DATA_BLOCK "DB_M256A_Scada"
{ DB_Accessible_From_OPC_UA := 'FALSE' ;
 DB_Accessible_From_Webserver := 'FALSE' ;
 S7_Optimized_Access := 'FALSE' }
VERSION : 0.1
NON_RETAIN
   STRUCT
      tAlm : Struct   // HMI Alarms
         tE { ExternalWritable := 'False'} : Struct
            x0 { ExternalWritable := 'False'} : Bool;
            x1 { ExternalWritable := 'False'} : Bool;
            x2 { ExternalWritable := 'False'} : Bool;
            x3 { ExternalWritable := 'False'} : Bool;
            x4 { ExternalWritable := 'False'} : Bool;
            x5 { ExternalWritable := 'False'} : Bool;
            x6 { ExternalWritable := 'False'} : Bool;
            x7 { ExternalWritable := 'False'} : Bool;
            x8 { ExternalWritable := 'False'} : Bool;
            x9 { ExternalWritable := 'False'} : Bool;
            x10 { ExternalWritable := 'False'} : Bool;
            x11 { ExternalWritable := 'False'} : Bool;
            x12 { ExternalWritable := 'False'} : Bool;
            x13 { ExternalWritable := 'False'} : Bool;
            x14 { ExternalWritable := 'False'} : Bool;
            x15 { ExternalWritable := 'False'} : Bool;
            x16 { ExternalWritable := 'False'} : Bool;
            x17 { ExternalWritable := 'False'} : Bool;
            x18 { ExternalWritable := 'False'} : Bool;
            x19 { ExternalWritable := 'False'} : Bool;
            x20 { ExternalWritable := 'False'} : Bool;
            x21 { ExternalWritable := 'False'} : Bool;
            x22 { ExternalWritable := 'False'} : Bool;
            x23 { ExternalWritable := 'False'} : Bool;
            x24 { ExternalWritable := 'False'} : Bool;
            x25 { ExternalWritable := 'False'} : Bool;
            x26 { ExternalWritable := 'False'} : Bool;
            x27 { ExternalWritable := 'False'} : Bool;
            x28 { ExternalWritable := 'False'} : Bool;
            x29 { ExternalWritable := 'False'} : Bool;
            x30 { ExternalWritable := 'False'} : Bool;
            x31 { ExternalWritable := 'False'} : Bool;
         END_STRUCT;
         tS { ExternalWritable := 'False'} : Struct
            tS0 { ExternalWritable := 'False'} : Struct
               x0 { ExternalWritable := 'False'} : Bool;   // Head#1 carriage not in working position
               x1 { ExternalWritable := 'False'} : Bool;   //
               x2 { ExternalWritable := 'False'} : Bool;
               x3 { ExternalWritable := 'False'} : Bool;
               x4 { ExternalWritable := 'False'} : Bool;
               x5 { ExternalWritable := 'False'} : Bool;
               x6 { ExternalWritable := 'False'} : Bool;
               x7 { ExternalWritable := 'False'} : Bool;
               x8 { ExternalWritable := 'False'} : Bool;
               x9 { ExternalWritable := 'False'} : Bool;   // Head#2carriage not in working position
               x10 { ExternalWritable := 'False'} : Bool;
               x11 { ExternalWritable := 'False'} : Bool;
               x12 { ExternalWritable := 'False'} : Bool;
               x13 { ExternalWritable := 'False'} : Bool;
               x14 { ExternalWritable := 'False'} : Bool;
               x15 { ExternalWritable := 'False'} : Bool;
               x16 { ExternalWritable := 'False'} : Bool;
               x17 { ExternalWritable := 'False'} : Bool;
               x18 { ExternalWritable := 'False'} : Bool;   // Head#3carriage not in working position
               x19 { ExternalWritable := 'False'} : Bool;
               x20 { ExternalWritable := 'False'} : Bool;
               x21 { ExternalWritable := 'False'} : Bool;
               x22 { ExternalWritable := 'False'} : Bool;
               x23 { ExternalWritable := 'False'} : Bool;
               x24 { ExternalWritable := 'False'} : Bool;
               x25 { ExternalWritable := 'False'} : Bool;
               x26 { ExternalWritable := 'False'} : Bool;
               x27 { ExternalWritable := 'False'} : Bool;
               x28 { ExternalWritable := 'False'} : Bool;
               x29 { ExternalWritable := 'False'} : Bool;
               x30 { ExternalWritable := 'False'} : Bool;
               x31 { ExternalWritable := 'False'} : Bool;
            END_STRUCT;
            tS1 { ExternalWritable := 'False'} : Struct
               x0 { ExternalWritable := 'False'} : Bool;   // Head#4carriage not in working position
               x1 { ExternalWritable := 'False'} : Bool;
               x2 { ExternalWritable := 'False'} : Bool;
               x3 { ExternalWritable := 'False'} : Bool;
               x4 { ExternalWritable := 'False'} : Bool;
               x5 { ExternalWritable := 'False'} : Bool;
               x6 { ExternalWritable := 'False'} : Bool;
               x7 { ExternalWritable := 'False'} : Bool;
               x8 { ExternalWritable := 'False'} : Bool;
               x9 { ExternalWritable := 'False'} : Bool;   // Head#5carriage not in working position
               x10 { ExternalWritable := 'False'} : Bool;
               x11 { ExternalWritable := 'False'} : Bool;
               x12 { ExternalWritable := 'False'} : Bool;
               x13 { ExternalWritable := 'False'} : Bool;
               x14 { ExternalWritable := 'False'} : Bool;
               x15 { ExternalWritable := 'False'} : Bool;
               x16 { ExternalWritable := 'False'} : Bool;
               x17 { ExternalWritable := 'False'} : Bool;
               x18 { ExternalWritable := 'False'} : Bool;   // Head#6carriage not in working position
               x19 { ExternalWritable := 'False'} : Bool;
               x20 { ExternalWritable := 'False'} : Bool;
               x21 { ExternalWritable := 'False'} : Bool;
               x22 { ExternalWritable := 'False'} : Bool;
               x23 { ExternalWritable := 'False'} : Bool;
               x24 { ExternalWritable := 'False'} : Bool;
               x25 { ExternalWritable := 'False'} : Bool;
               x26 { ExternalWritable := 'False'} : Bool;
               x27 { ExternalWritable := 'False'} : Bool;
               x28 { ExternalWritable := 'False'} : Bool;
               x29 { ExternalWritable := 'False'} : Bool;
               x30 { ExternalWritable := 'False'} : Bool;
               x31 { ExternalWritable := 'False'} : Bool;
            END_STRUCT;
            tS2 { ExternalWritable := 'False'} : Struct
               x0 { ExternalWritable := 'False'} : Bool;   // Head#7carriage not in working position
               x1 { ExternalWritable := 'False'} : Bool;
               x2 { ExternalWritable := 'False'} : Bool;
               x3 { ExternalWritable := 'False'} : Bool;
               x4 { ExternalWritable := 'False'} : Bool;
               x5 { ExternalWritable := 'False'} : Bool;
               x6 { ExternalWritable := 'False'} : Bool;
               x7 { ExternalWritable := 'False'} : Bool;
               x8 { ExternalWritable := 'False'} : Bool;
               x9 { ExternalWritable := 'False'} : Bool;   // Head#8carriage not in working position
               x10 { ExternalWritable := 'False'} : Bool;
               x11 { ExternalWritable := 'False'} : Bool;
               x12 { ExternalWritable := 'False'} : Bool;
               x13 { ExternalWritable := 'False'} : Bool;
               x14 { ExternalWritable := 'False'} : Bool;
               x15 { ExternalWritable := 'False'} : Bool;
               x16 { ExternalWritable := 'False'} : Bool;
               x17 { ExternalWritable := 'False'} : Bool;
               x18 { ExternalWritable := 'False'} : Bool;
               x19 { ExternalWritable := 'False'} : Bool;
               x20 { ExternalWritable := 'False'} : Bool;
               x21 { ExternalWritable := 'False'} : Bool;
               x22 { ExternalWritable := 'False'} : Bool;
               x23 { ExternalWritable := 'False'} : Bool;
               x24 { ExternalWritable := 'False'} : Bool;
               x25 { ExternalWritable := 'False'} : Bool;
               x26 { ExternalWritable := 'False'} : Bool;
               x27 { ExternalWritable := 'False'} : Bool;
               x28 { ExternalWritable := 'False'} : Bool;
               x29 { ExternalWritable := 'False'} : Bool;
               x30 { ExternalWritable := 'False'} : Bool;
               x31 { ExternalWritable := 'False'} : Bool;
            END_STRUCT;
            tS3 { ExternalWritable := 'False'} : Struct
               x0 { ExternalWritable := 'False'} : Bool;
               x1 { ExternalWritable := 'False'} : Bool;
               x2 { ExternalWritable := 'False'} : Bool;
               x3 { ExternalWritable := 'False'} : Bool;
               x4 { ExternalWritable := 'False'} : Bool;
               x5 { ExternalWritable := 'False'} : Bool;
               x6 { ExternalWritable := 'False'} : Bool;
               x7 { ExternalWritable := 'False'} : Bool;
               x8 { ExternalWritable := 'False'} : Bool;
               x9 { ExternalWritable := 'False'} : Bool;
               x10 { ExternalWritable := 'False'} : Bool;
               x11 { ExternalWritable := 'False'} : Bool;
               x12 { ExternalWritable := 'False'} : Bool;
               x13 { ExternalWritable := 'False'} : Bool;
               x14 { ExternalWritable := 'False'} : Bool;
               x15 { ExternalWritable := 'False'} : Bool;
               x16 { ExternalWritable := 'False'} : Bool;
               x17 { ExternalWritable := 'False'} : Bool;
               x18 { ExternalWritable := 'False'} : Bool;
               x19 { ExternalWritable := 'False'} : Bool;
               x20 { ExternalWritable := 'False'} : Bool;
               x21 { ExternalWritable := 'False'} : Bool;
               x22 { ExternalWritable := 'False'} : Bool;
               x23 { ExternalWritable := 'False'} : Bool;
               x24 { ExternalWritable := 'False'} : Bool;
               x25 { ExternalWritable := 'False'} : Bool;
               x26 { ExternalWritable := 'False'} : Bool;
               x27 { ExternalWritable := 'False'} : Bool;
               x28 { ExternalWritable := 'False'} : Bool;
               x29 { ExternalWritable := 'False'} : Bool;
               x30 { ExternalWritable := 'False'} : Bool;
               x31 { ExternalWritable := 'False'} : Bool;
            END_STRUCT;
         END_STRUCT;
         tF { ExternalWritable := 'False'} : Struct
            x0 { ExternalWritable := 'False'} : Bool;
            x1 { ExternalWritable := 'False'} : Bool;
            x2 { ExternalWritable := 'False'} : Bool;
            x3 { ExternalWritable := 'False'} : Bool;
            x4 { ExternalWritable := 'False'} : Bool;
            x5 { ExternalWritable := 'False'} : Bool;
            x6 { ExternalWritable := 'False'} : Bool;
            x7 { ExternalWritable := 'False'} : Bool;
            x8 { ExternalWritable := 'False'} : Bool;
            x9 { ExternalWritable := 'False'} : Bool;
            x10 { ExternalWritable := 'False'} : Bool;
            x11 { ExternalWritable := 'False'} : Bool;
            x12 { ExternalWritable := 'False'} : Bool;
            x13 { ExternalWritable := 'False'} : Bool;
            x14 { ExternalWritable := 'False'} : Bool;
            x15 { ExternalWritable := 'False'} : Bool;
            x16 { ExternalWritable := 'False'} : Bool;
            x17 { ExternalWritable := 'False'} : Bool;
            x18 { ExternalWritable := 'False'} : Bool;
            x19 { ExternalWritable := 'False'} : Bool;
            x20 { ExternalWritable := 'False'} : Bool;
            x21 { ExternalWritable := 'False'} : Bool;
            x22 { ExternalWritable := 'False'} : Bool;
            x23 { ExternalWritable := 'False'} : Bool;
            x24 { ExternalWritable := 'False'} : Bool;
            x25 { ExternalWritable := 'False'} : Bool;
            x26 { ExternalWritable := 'False'} : Bool;
            x27 { ExternalWritable := 'False'} : Bool;
            x28 { ExternalWritable := 'False'} : Bool;
            x29 { ExternalWritable := 'False'} : Bool;
            x30 { ExternalWritable := 'False'} : Bool;
            x31 { ExternalWritable := 'False'} : Bool;
         END_STRUCT;
         tW { ExternalWritable := 'False'} : Struct
            x0 { ExternalWritable := 'False'} : Bool;
            x1 { ExternalWritable := 'False'} : Bool;
            x2 { ExternalWritable := 'False'} : Bool;
            x3 { ExternalWritable := 'False'} : Bool;
            x4 { ExternalWritable := 'False'} : Bool;
            x5 { ExternalWritable := 'False'} : Bool;
            x6 { ExternalWritable := 'False'} : Bool;
            x7 { ExternalWritable := 'False'} : Bool;
            x8 { ExternalWritable := 'False'} : Bool;
            x9 { ExternalWritable := 'False'} : Bool;
            x10 { ExternalWritable := 'False'} : Bool;
            x11 { ExternalWritable := 'False'} : Bool;
            x12 { ExternalWritable := 'False'} : Bool;
            x13 { ExternalWritable := 'False'} : Bool;
            x14 { ExternalWritable := 'False'} : Bool;
            x15 { ExternalWritable := 'False'} : Bool;
            x16 { ExternalWritable := 'False'} : Bool;
            x17 { ExternalWritable := 'False'} : Bool;
            x18 { ExternalWritable := 'False'} : Bool;
            x19 { ExternalWritable := 'False'} : Bool;
            x20 { ExternalWritable := 'False'} : Bool;
            x21 { ExternalWritable := 'False'} : Bool;
            x22 { ExternalWritable := 'False'} : Bool;
            x23 { ExternalWritable := 'False'} : Bool;
            x24 { ExternalWritable := 'False'} : Bool;
            x25 { ExternalWritable := 'False'} : Bool;
            x26 { ExternalWritable := 'False'} : Bool;
            x27 { ExternalWritable := 'False'} : Bool;
            x28 { ExternalWritable := 'False'} : Bool;
            x29 { ExternalWritable := 'False'} : Bool;
            x30 { ExternalWritable := 'False'} : Bool;
            x31 { ExternalWritable := 'False'} : Bool;
         END_STRUCT;
      END_STRUCT;
      tHMR { ExternalWritable := 'False'} : Struct   // HMI Read
         xSpare0 { ExternalWritable := 'False'} : Bool;   //
         xSpare1 { ExternalWritable := 'False'} : Bool;
         xSpare2 { ExternalWritable := 'False'} : Bool;
         xSpare3 { ExternalWritable := 'False'} : Bool;
         xSpare4 { ExternalWritable := 'False'} : Bool;
         xSpare5 { ExternalWritable := 'False'} : Bool;
         xSpare6 { ExternalWritable := 'False'} : Bool;
         xSpare7 { ExternalWritable := 'False'} : Bool;
         xSpare8 { ExternalWritable := 'False'} : Bool;
         xSpare9 { ExternalWritable := 'False'} : Bool;
         xSpare10 { ExternalWritable := 'False'} : Bool;
         xSpare11 { ExternalWritable := 'False'} : Bool;
         xSpare12 { ExternalWritable := 'False'} : Bool;
         xSpare13 { ExternalWritable := 'False'} : Bool;
         xSpare14 { ExternalWritable := 'False'} : Bool;
         xSpare15 { ExternalWritable := 'False'} : Bool;
         xSpare16 { ExternalWritable := 'False'} : Bool;
         xSpare17 { ExternalWritable := 'False'} : Bool;
         xSpare18 { ExternalWritable := 'False'} : Bool;
         xSpare19 { ExternalWritable := 'False'} : Bool;
         xSpare20 { ExternalWritable := 'False'} : Bool;
         xSpare21 { ExternalWritable := 'False'} : Bool;
         xSpare22 { ExternalWritable := 'False'} : Bool;
         xSpare23 { ExternalWritable := 'False'} : Bool;
         xSpare24 { ExternalWritable := 'False'} : Bool;
         xSpare25 { ExternalWritable := 'False'} : Bool;
         xSpare26 { ExternalWritable := 'False'} : Bool;
         xSpare27 { ExternalWritable := 'False'} : Bool;
         xSpare28 { ExternalWritable := 'False'} : Bool;
         xSpare29 { ExternalWritable := 'False'} : Bool;
         xSpare30 { ExternalWritable := 'False'} : Bool;
         xSpare31 { ExternalWritable := 'False'} : Bool;
         xSpare { ExternalWritable := 'False'} : Array[0..15] of Bool;
         iSpare0 { ExternalWritable := 'False'} : Int;
         iSpare1 { ExternalWritable := 'False'} : Int;
         iSpare2 { ExternalWritable := 'False'} : Int;
         iSpare3 { ExternalWritable := 'False'} : Int;
         iSpare4 { ExternalWritable := 'False'} : Int;
         iSpare5 { ExternalWritable := 'False'} : Int;
         iSpare6 { ExternalWritable := 'False'} : Int;
         iSpare7 { ExternalWritable := 'False'} : Int;
         iSpare8 { ExternalWritable := 'False'} : Int;
         iSpare9 { ExternalWritable := 'False'} : Int;
         iSpare10 { ExternalWritable := 'False'} : Int;
         iSpare11 { ExternalWritable := 'False'} : Int;
         iSpare12 { ExternalWritable := 'False'} : Int;
         iSpare13 { ExternalWritable := 'False'} : Int;
         iSpare14 { ExternalWritable := 'False'} : Int;
         iSpare15 { ExternalWritable := 'False'} : Int;
         iSpare16 { ExternalWritable := 'False'} : Int;
         dHeadStatus_H1 { ExternalWritable := 'False'} : DInt;   // Head#1 arming status (1=Up 3=Down 7=Anomaly) {x|x|x|x|O}
         dHeadStatus_H2 { ExternalWritable := 'False'} : DInt;   // Head#2 arming status (1=Up 3=Down 7=Anomaly) {x|x|x|x|O}
         dHeadStatus_H3 { ExternalWritable := 'False'} : DInt;   // Head#3 arming status (1=Up 3=Down 7=Anomaly) {x|x|x|x|O}
         dHeadStatus_H4 { ExternalWritable := 'False'} : DInt;   // Head#4 arming status (1=Up 3=Down 7=Anomaly) {x|x|x|x|O}
         dHeadStatus_H5 { ExternalWritable := 'False'} : DInt;   // Head#5 arming status (1=Up 3=Down 7=Anomaly) {x|x|x|x|O}
         dHeadStatus_H6 { ExternalWritable := 'False'} : DInt;   // Head#6 arming status (1=Up 3=Down 7=Anomaly) {x|x|x|x|O}
         dHeadStatus_H7 { ExternalWritable := 'False'} : DInt;   // Head#7 arming status (1=Up 3=Down 7=Anomaly) {x|x|x|x|O}
         dHeadStatus_H8 { ExternalWritable := 'False'} : DInt;   // Head#8 arming status (1=Up 3=Down 7=Anomaly) {x|x|x|x|O}
         dSpare8 { ExternalWritable := 'False'} : DInt;
         dSpare9 { ExternalWritable := 'False'} : DInt;
         dSpare10 { ExternalWritable := 'False'} : DInt;
         dSpare11 { ExternalWritable := 'False'} : DInt;
         dSpare12 { ExternalWritable := 'False'} : DInt;
         dSpare13 { ExternalWritable := 'False'} : DInt;
         dSpare14 { ExternalWritable := 'False'} : DInt;
         dSpare15 { ExternalWritable := 'False'} : DInt;
         dSpare { ExternalWritable := 'False'} : Array[0..15] of DInt;
         rSpare0 { ExternalWritable := 'False'} : Real;
         rSpare1 { ExternalWritable := 'False'} : Real;
         rSpare2 { ExternalWritable := 'False'} : Real;
         rSpare3 { ExternalWritable := 'False'} : Real;
         rSpare4 { ExternalWritable := 'False'} : Real;
         rSpare5 { ExternalWritable := 'False'} : Real;
         rSpare6 { ExternalWritable := 'False'} : Real;
         rSpare7 { ExternalWritable := 'False'} : Real;
         rSpare8 { ExternalWritable := 'False'} : Real;
         tManCmd { ExternalWritable := 'False'} : Struct
            xMan_DescentFdbk_H1 { ExternalWritable := 'False'} : Bool;   // Head #1 manual descent feedback {x|x|x|x|O}
            xMan_RiseFdbk_H1 { ExternalWritable := 'False'} : Bool;   // Head #1 manual rise feedback {x|x|x|x|O}
            xMan_DescentFdbk_H2 { ExternalWritable := 'False'} : Bool;   // Head #2 manual descent feedback {x|x|x|x|O}
            xMan_RiseFdbk_H2 { ExternalWritable := 'False'} : Bool;   // Head #2 manual rise feedback {x|x|x|x|O}
            xMan_DescentFdbk_H3 { ExternalWritable := 'False'} : Bool;   // Head #3 manual descent feedback {x|x|x|x|O}
            xMan_RiseFdbk_H3 { ExternalWritable := 'False'} : Bool;   // Head #3 manual rise feedback {x|x|x|x|O}
            xMan_DescentFdbk_H4 { ExternalWritable := 'False'} : Bool;   // Head #4 manual descent feedback {x|x|x|x|O}
            xMan_RiseFdbk_H4 { ExternalWritable := 'False'} : Bool;   // Head #4 manual rise feedback {x|x|x|x|O}
            xMan_DescentFdbk_H5 { ExternalWritable := 'False'} : Bool;   // Head #5 manual descent feedback {x|x|x|x|O}
            xMan_RiseFdbk_H5 { ExternalWritable := 'False'} : Bool;   // Head #5 manual rise feedback {x|x|x|x|O}
            xMan_DescentFdbk_H6 { ExternalWritable := 'False'} : Bool;   // Head #6 manual descent feedback {x|x|x|x|O}
            xMan_RiseFdbk_H6 { ExternalWritable := 'False'} : Bool;   // Head #6 manual rise feedback {x|x|x|x|O}
            xMan_DescentFdbk_H7 { ExternalWritable := 'False'} : Bool;   // Head #7 manual descent feedback {x|x|x|x|O}
            xMan_RiseFdbk_H7 { ExternalWritable := 'False'} : Bool;   // Head #7 manual rise feedback {x|x|x|x|O}
            xMan_DescentFdbk_H8 { ExternalWritable := 'False'} : Bool;   // Head #8 manual descent feedback {x|x|x|x|O}
            xMan_RiseFdbk_H8 { ExternalWritable := 'False'} : Bool;   // Head #8 manual rise feedback {x|x|x|x|O}
            xSpare { ExternalWritable := 'False'} : Array[0..15] of Bool;
         END_STRUCT;
      END_STRUCT;
      tHMW : Struct   // HMI Write
         xSpare0 : Bool;
         xSpare1 : Bool;
         xSpare2 : Bool;
         xSpare3 : Bool;
         xSpare4 : Bool;
         xSpare5 : Bool;
         xSpare6 : Bool;
         xSpare7 : Bool;
         xSpare8 : Bool;
         xSpare9 : Bool;
         xSpare10 : Bool;
         xSpare11 : Bool;
         xSpare12 : Bool;
         xSpare13 : Bool;
         xSpare14 : Bool;
         xSpare15 : Bool;
         xSpare16 : Bool;
         xSpare17 : Bool;
         xSpare18 : Bool;
         xSpare19 : Bool;
         xSpare20 : Bool;
         xSpare21 : Bool;
         xSpare22 : Bool;
         xSpare23 : Bool;
         xSpare24 : Bool;
         xSpare25 : Bool;
         xSpare26 : Bool;
         xSpare27 : Bool;
         xSpare28 : Bool;
         xSpare29 : Bool;
         xSpare30 : Bool;
         xSpare31 : Bool;
         xSpare : Array[0..15] of Bool;
         iSpare0 : Int;
         iSpare1 : Int;
         iSpare2 : Int;
         iSpare3 : Int;
         iSpare4 : Int;
         iSpare5 : Int;
         iSpare6 : Int;
         iSpare7 : Int;
         iSpare8 : Int;
         iSpare9 : Int;
         iSpare10 : Int;
         iSpare11 : Int;
         iSpare12 : Int;
         iSpare13 : Int;
         iSpare14 : Int;
         iSpare15 : Int;
         iSpare16 : Int;
         dRaiseReactTime_ms_H1 : DInt;   // Head#1 raise reaction time [ms] {ms|s|-200|200|M}
         dDescentReactTime_ms_H1 : DInt;   // Head#1 descent reaction time [ms] {ms|s|0|3000|M}
         dRaiseReactTime_ms_H2 : DInt;   // Head#2 raise reaction time [ms] {ms|s|-200|200|M}
         dDescentReactTime_ms_H2 : DInt;   // Head#2 descent reaction time [ms] {ms|s|0|3000|M}
         dRaiseReactTime_ms_H3 : DInt;   // Head#3 raise reaction time [ms] {ms|s|-200|200|M}
         dDescentReactTime_ms_H3 : DInt;   // Head#3 descent reaction time [ms] {ms|s|0|3000|M}
         dRaiseReactTime_ms_H4 : DInt;   // Head#4 raise reaction time [ms] {ms|s|-200|200|M}
         dDescentReactTime_ms_H4 : DInt;   // Head#4 descent reaction time [ms] {ms|s|0|3000|M}
         dRaiseReactTime_ms_H5 : DInt;   // Head#5raise reaction time [ms] {ms|s|-200|200|M}
         dDescentReactTime_ms_H5 : DInt;   // Head#5descent reaction time [ms] {ms|s|0|3000|M}
         dRaiseReactTime_ms_H6 : DInt;   // Head#6 raise reaction time [ms] {ms|s|-200|200|M}
         dDescentReactTime_ms_H6 : DInt;   // Head#6 descent reaction time [ms] {ms|s|0|3000|M}
         dRaiseReactTime_ms_H7 : DInt;   // Head#7 raise reaction time [ms] {ms|s|-200|200|M}
         dDescentReactTime_ms_H7 : DInt;   // Head#7 descent reaction time [ms] {ms|s|0|3000|M}
         dRaiseReactTime_ms_H8 : DInt;   // Head#8 raise reaction time [ms] {ms|s|-200|200|M}
         dDescentReactTime_ms_H8 : DInt;   // Head#8 descent reaction time [ms] {ms|s|0|3000|M}
         dSpare16 : DInt;
         dSpare17 : DInt;
         dSpare18 : DInt;
         dSpare19 : DInt;
         dSpare20 : DInt;
         dSpare21 : DInt;
         dSpare22 : DInt;
         dSpare23 : DInt;
         dSpare24 : DInt;
         dSpare25 : DInt;
         dSpare26 : DInt;
         dSpare27 : DInt;
         dSpare28 : DInt;
         dSpare29 : DInt;
         dSpare30 : DInt;
         dSpare31 : DInt;
         dSpare32 : DInt;
         dSpare33 : DInt;
         dSpare34 : DInt;
         dSpare35 : DInt;
         dSpare36 : DInt;
         dSpare37 : DInt;
         dSpare38 : DInt;
         dSpare39 : DInt;
         dSpare { ExternalWritable := 'False'} : Array[0..19] of DInt;
         rSpare0 : Real;
         rSpare1 : Real;
         rSpare2 : Real;
         rSpare3 : Real;
         rSpare4 : Real;
         rSpare5 : Real;
         rSpare6 : Real;
         rSpare7 : Real;
         rSpare8 : Real;
         tManCmd : Struct
            xManDescent_H1 : Bool;   // Head #1 manual Descent {x|x|x|x|O}
            xManRise_H1 : Bool;   // Head #1 manual rise {x|x|x|x|O}
            xManRise_H2 : Bool;   // Head #2 manual rise {x|x|x|x|O}
            xManDescent_H2 : Bool;   // Head #2 manual Descent {x|x|x|x|O}
            xManRise_H3 : Bool;   // Head #3 manual rise {x|x|x|x|O}
            xManDescent_H3 : Bool;   // Head #3 manual Descent {x|x|x|x|O}
            xManRise_H4 : Bool;   // Head #4 manual rise {x|x|x|x|O}
            xManDescent_H4 : Bool;   // Head #4 manual Descent {x|x|x|x|O}
            xManRise_H5 : Bool;   // Head #5 manual rise {x|x|x|x|O}
            xManDescent_H5 : Bool;   // Head #5 manual Descent {x|x|x|x|O}
            xManRise_H6 : Bool;   // Head #6 manual rise {x|x|x|x|O}
            xManDescent_H6 : Bool;   // Head #6 manual Descent {x|x|x|x|O}
            xManRise_H7 : Bool;   // Head #7 manual rise {x|x|x|x|O}
            xManDescent_H7 : Bool;   // Head #7 manual Descent {x|x|x|x|O}
            xManRise_H8 : Bool;   // Head #8 manual rise {x|x|x|x|O}
            xManDescent_H8 : Bool;   // Head #8 manual Descent {x|x|x|x|O}
            xSpare16 : Bool;
            xSpare17 : Bool;
            xSpare18 : Bool;
            xSpare19 : Bool;
            xSpare20 : Bool;
            xSpare21 : Bool;
            xSpare22 : Bool;
            xSpare23 : Bool;
            xSpare24 : Bool;
            xSpare25 : Bool;
            xSpare26 : Bool;
            xSpare27 : Bool;
            xSpare28 : Bool;
            xSpare29 : Bool;
            xSpare30 : Bool;
            xSpare31 : Bool;
         END_STRUCT;
      END_STRUCT;
   END_STRUCT;


BEGIN
   tHMR.xSpare0 := FALSE;
   tHMR.xSpare15 := FALSE;
   tHMR.dSpare8 := 0;
   tHMR.dSpare9 := 0;
   tHMR.dSpare10 := 0;
   tHMR.dSpare11 := 0;
   tHMW.xSpare0 := FALSE;
   tHMW.xSpare1 := FALSE;
   tHMW.xSpare2 := FALSE;
   tHMW.xSpare3 := FALSE;
   tHMW.xSpare4 := FALSE;
   tHMW.xSpare5 := FALSE;
   tHMW.xSpare6 := FALSE;
   tHMW.xSpare7 := FALSE;
   tHMW.xSpare8 := FALSE;
   tHMW.xSpare14 := FALSE;
   tHMW.xSpare15 := FALSE;
   tHMW.xSpare16 := TRUE;
   tHMW.xSpare17 := TRUE;
   tHMW.xSpare18 := TRUE;
   tHMW.xSpare19 := TRUE;
   tHMW.xSpare20 := TRUE;
   tHMW.xSpare21 := TRUE;
   tHMW.xSpare22 := TRUE;
   tHMW.xSpare23 := TRUE;
   tHMW.iSpare16 := 0;

END_DATA_BLOCK

DATA_BLOCK "DB_M256F_Scada"
{ DB_Accessible_From_OPC_UA := 'FALSE' ;
 DB_Accessible_From_Webserver := 'FALSE' ;
 S7_Optimized_Access := 'FALSE' }
VERSION : 0.1
NON_RETAIN
   STRUCT
      tAlm : Struct   // HMI Alarms
         tE { ExternalWritable := 'False'} : Struct
            x0 { ExternalWritable := 'False'} : Bool;
            x1 { ExternalWritable := 'False'} : Bool;
            x2 { ExternalWritable := 'False'} : Bool;
            x3 { ExternalWritable := 'False'} : Bool;
            x4 { ExternalWritable := 'False'} : Bool;
            x5 { ExternalWritable := 'False'} : Bool;
            x6 { ExternalWritable := 'False'} : Bool;
            x7 { ExternalWritable := 'False'} : Bool;
            x8 { ExternalWritable := 'False'} : Bool;
            x9 { ExternalWritable := 'False'} : Bool;
            x10 { ExternalWritable := 'False'} : Bool;
            x11 { ExternalWritable := 'False'} : Bool;
            x12 { ExternalWritable := 'False'} : Bool;
            x13 { ExternalWritable := 'False'} : Bool;
            x14 { ExternalWritable := 'False'} : Bool;
            x15 { ExternalWritable := 'False'} : Bool;
            x16 { ExternalWritable := 'False'} : Bool;
            x17 { ExternalWritable := 'False'} : Bool;
            x18 { ExternalWritable := 'False'} : Bool;
            x19 { ExternalWritable := 'False'} : Bool;
            x20 { ExternalWritable := 'False'} : Bool;
            x21 { ExternalWritable := 'False'} : Bool;
            x22 { ExternalWritable := 'False'} : Bool;
            x23 { ExternalWritable := 'False'} : Bool;
            x24 { ExternalWritable := 'False'} : Bool;
            x25 { ExternalWritable := 'False'} : Bool;
            x26 { ExternalWritable := 'False'} : Bool;
            x27 { ExternalWritable := 'False'} : Bool;
            x28 { ExternalWritable := 'False'} : Bool;
            x29 { ExternalWritable := 'False'} : Bool;
            x30 { ExternalWritable := 'False'} : Bool;
            x31 { ExternalWritable := 'False'} : Bool;
         END_STRUCT;
         tS { ExternalWritable := 'False'} : Struct
            tS0 { ExternalWritable := 'False'} : Struct
               x0 { ExternalWritable := 'False'} : Bool;
               x1 { ExternalWritable := 'False'} : Bool;
               x2 { ExternalWritable := 'False'} : Bool;
               x3 { ExternalWritable := 'False'} : Bool;
               x4 { ExternalWritable := 'False'} : Bool;
               x5 { ExternalWritable := 'False'} : Bool;
               x6 { ExternalWritable := 'False'} : Bool;
               x7 { ExternalWritable := 'False'} : Bool;
               x8 { ExternalWritable := 'False'} : Bool;
               x9 { ExternalWritable := 'False'} : Bool;
               x10 { ExternalWritable := 'False'} : Bool;
               x11 { ExternalWritable := 'False'} : Bool;
               x12 { ExternalWritable := 'False'} : Bool;
               x13 { ExternalWritable := 'False'} : Bool;
               x14 { ExternalWritable := 'False'} : Bool;
               x15 { ExternalWritable := 'False'} : Bool;
               x16 { ExternalWritable := 'False'} : Bool;
               x17 { ExternalWritable := 'False'} : Bool;
               x18 { ExternalWritable := 'False'} : Bool;
               x19 { ExternalWritable := 'False'} : Bool;
               x20 { ExternalWritable := 'False'} : Bool;
               x21 { ExternalWritable := 'False'} : Bool;
               x22 { ExternalWritable := 'False'} : Bool;
               x23 { ExternalWritable := 'False'} : Bool;
               x24 { ExternalWritable := 'False'} : Bool;
               x25 { ExternalWritable := 'False'} : Bool;
               x26 { ExternalWritable := 'False'} : Bool;
               x27 { ExternalWritable := 'False'} : Bool;
               x28 { ExternalWritable := 'False'} : Bool;
               x29 { ExternalWritable := 'False'} : Bool;
               x30 { ExternalWritable := 'False'} : Bool;
               x31 { ExternalWritable := 'False'} : Bool;
            END_STRUCT;
            tS1 { ExternalWritable := 'False'} : Struct
               x0 { ExternalWritable := 'False'} : Bool;
               x1 { ExternalWritable := 'False'} : Bool;
               x2 { ExternalWritable := 'False'} : Bool;
               x3 { ExternalWritable := 'False'} : Bool;
               x4 { ExternalWritable := 'False'} : Bool;
               x5 { ExternalWritable := 'False'} : Bool;
               x6 { ExternalWritable := 'False'} : Bool;
               x7 { ExternalWritable := 'False'} : Bool;
               x8 { ExternalWritable := 'False'} : Bool;
               x9 { ExternalWritable := 'False'} : Bool;
               x10 { ExternalWritable := 'False'} : Bool;
               x11 { ExternalWritable := 'False'} : Bool;
               x12 { ExternalWritable := 'False'} : Bool;
               x13 { ExternalWritable := 'False'} : Bool;
               x14 { ExternalWritable := 'False'} : Bool;
               x15 { ExternalWritable := 'False'} : Bool;
               x16 { ExternalWritable := 'False'} : Bool;
               x17 { ExternalWritable := 'False'} : Bool;
               x18 { ExternalWritable := 'False'} : Bool;
               x19 { ExternalWritable := 'False'} : Bool;
               x20 { ExternalWritable := 'False'} : Bool;
               x21 { ExternalWritable := 'False'} : Bool;
               x22 { ExternalWritable := 'False'} : Bool;
               x23 { ExternalWritable := 'False'} : Bool;
               x24 { ExternalWritable := 'False'} : Bool;
               x25 { ExternalWritable := 'False'} : Bool;
               x26 { ExternalWritable := 'False'} : Bool;
               x27 { ExternalWritable := 'False'} : Bool;
               x28 { ExternalWritable := 'False'} : Bool;
               x29 { ExternalWritable := 'False'} : Bool;
               x30 { ExternalWritable := 'False'} : Bool;
               x31 { ExternalWritable := 'False'} : Bool;
            END_STRUCT;
            tS2 { ExternalWritable := 'False'} : Struct
               x0 { ExternalWritable := 'False'} : Bool;
               x1 { ExternalWritable := 'False'} : Bool;
               x2 { ExternalWritable := 'False'} : Bool;
               x3 { ExternalWritable := 'False'} : Bool;
               x4 { ExternalWritable := 'False'} : Bool;
               x5 { ExternalWritable := 'False'} : Bool;
               x6 { ExternalWritable := 'False'} : Bool;
               x7 { ExternalWritable := 'False'} : Bool;
               x8 { ExternalWritable := 'False'} : Bool;
               x9 { ExternalWritable := 'False'} : Bool;
               x10 { ExternalWritable := 'False'} : Bool;
               x11 { ExternalWritable := 'False'} : Bool;
               x12 { ExternalWritable := 'False'} : Bool;
               x13 { ExternalWritable := 'False'} : Bool;
               x14 { ExternalWritable := 'False'} : Bool;
               x15 { ExternalWritable := 'False'} : Bool;
               x16 { ExternalWritable := 'False'} : Bool;
               x17 { ExternalWritable := 'False'} : Bool;
               x18 { ExternalWritable := 'False'} : Bool;
               x19 { ExternalWritable := 'False'} : Bool;
               x20 { ExternalWritable := 'False'} : Bool;
               x21 { ExternalWritable := 'False'} : Bool;
               x22 { ExternalWritable := 'False'} : Bool;
               x23 { ExternalWritable := 'False'} : Bool;
               x24 { ExternalWritable := 'False'} : Bool;
               x25 { ExternalWritable := 'False'} : Bool;
               x26 { ExternalWritable := 'False'} : Bool;
               x27 { ExternalWritable := 'False'} : Bool;
               x28 { ExternalWritable := 'False'} : Bool;
               x29 { ExternalWritable := 'False'} : Bool;
               x30 { ExternalWritable := 'False'} : Bool;
               x31 { ExternalWritable := 'False'} : Bool;
            END_STRUCT;
            tS3 { ExternalWritable := 'False'} : Struct
               x0 { ExternalWritable := 'False'} : Bool;
               x1 { ExternalWritable := 'False'} : Bool;
               x2 { ExternalWritable := 'False'} : Bool;
               x3 { ExternalWritable := 'False'} : Bool;
               x4 { ExternalWritable := 'False'} : Bool;
               x5 { ExternalWritable := 'False'} : Bool;
               x6 { ExternalWritable := 'False'} : Bool;
               x7 { ExternalWritable := 'False'} : Bool;
               x8 { ExternalWritable := 'False'} : Bool;
               x9 { ExternalWritable := 'False'} : Bool;
               x10 { ExternalWritable := 'False'} : Bool;
               x11 { ExternalWritable := 'False'} : Bool;
               x12 { ExternalWritable := 'False'} : Bool;
               x13 { ExternalWritable := 'False'} : Bool;
               x14 { ExternalWritable := 'False'} : Bool;
               x15 { ExternalWritable := 'False'} : Bool;
               x16 { ExternalWritable := 'False'} : Bool;
               x17 { ExternalWritable := 'False'} : Bool;
               x18 { ExternalWritable := 'False'} : Bool;
               x19 { ExternalWritable := 'False'} : Bool;
               x20 { ExternalWritable := 'False'} : Bool;
               x21 { ExternalWritable := 'False'} : Bool;
               x22 { ExternalWritable := 'False'} : Bool;
               x23 { ExternalWritable := 'False'} : Bool;
               x24 { ExternalWritable := 'False'} : Bool;
               x25 { ExternalWritable := 'False'} : Bool;
               x26 { ExternalWritable := 'False'} : Bool;
               x27 { ExternalWritable := 'False'} : Bool;
               x28 { ExternalWritable := 'False'} : Bool;
               x29 { ExternalWritable := 'False'} : Bool;
               x30 { ExternalWritable := 'False'} : Bool;
               x31 { ExternalWritable := 'False'} : Bool;
            END_STRUCT;
         END_STRUCT;
         tF { ExternalWritable := 'False'} : Struct
            x0 { ExternalWritable := 'False'} : Bool;
            x1 { ExternalWritable := 'False'} : Bool;
            x2 { ExternalWritable := 'False'} : Bool;
            x3 { ExternalWritable := 'False'} : Bool;
            x4 { ExternalWritable := 'False'} : Bool;
            x5 { ExternalWritable := 'False'} : Bool;
            x6 { ExternalWritable := 'False'} : Bool;
            x7 { ExternalWritable := 'False'} : Bool;
            x8 { ExternalWritable := 'False'} : Bool;
            x9 { ExternalWritable := 'False'} : Bool;
            x10 { ExternalWritable := 'False'} : Bool;
            x11 { ExternalWritable := 'False'} : Bool;
            x12 { ExternalWritable := 'False'} : Bool;
            x13 { ExternalWritable := 'False'} : Bool;
            x14 { ExternalWritable := 'False'} : Bool;
            x15 { ExternalWritable := 'False'} : Bool;
            x16 { ExternalWritable := 'False'} : Bool;
            x17 { ExternalWritable := 'False'} : Bool;
            x18 { ExternalWritable := 'False'} : Bool;
            x19 { ExternalWritable := 'False'} : Bool;
            x20 { ExternalWritable := 'False'} : Bool;
            x21 { ExternalWritable := 'False'} : Bool;
            x22 { ExternalWritable := 'False'} : Bool;
            x23 { ExternalWritable := 'False'} : Bool;
            x24 { ExternalWritable := 'False'} : Bool;
            x25 { ExternalWritable := 'False'} : Bool;
            x26 { ExternalWritable := 'False'} : Bool;
            x27 { ExternalWritable := 'False'} : Bool;
            x28 { ExternalWritable := 'False'} : Bool;
            x29 { ExternalWritable := 'False'} : Bool;
            x30 { ExternalWritable := 'False'} : Bool;
            x31 { ExternalWritable := 'False'} : Bool;
         END_STRUCT;
         tW { ExternalWritable := 'False'} : Struct
            x0 { ExternalWritable := 'False'} : Bool;
            x1 { ExternalWritable := 'False'} : Bool;
            x2 { ExternalWritable := 'False'} : Bool;
            x3 { ExternalWritable := 'False'} : Bool;
            x4 { ExternalWritable := 'False'} : Bool;
            x5 { ExternalWritable := 'False'} : Bool;
            x6 { ExternalWritable := 'False'} : Bool;
            x7 { ExternalWritable := 'False'} : Bool;
            x8 { ExternalWritable := 'False'} : Bool;
            x9 { ExternalWritable := 'False'} : Bool;
            x10 { ExternalWritable := 'False'} : Bool;
            x11 { ExternalWritable := 'False'} : Bool;
            x12 { ExternalWritable := 'False'} : Bool;
            x13 { ExternalWritable := 'False'} : Bool;
            x14 { ExternalWritable := 'False'} : Bool;
            x15 { ExternalWritable := 'False'} : Bool;
            x16 { ExternalWritable := 'False'} : Bool;
            x17 { ExternalWritable := 'False'} : Bool;
            x18 { ExternalWritable := 'False'} : Bool;
            x19 { ExternalWritable := 'False'} : Bool;
            x20 { ExternalWritable := 'False'} : Bool;
            x21 { ExternalWritable := 'False'} : Bool;
            x22 { ExternalWritable := 'False'} : Bool;
            x23 { ExternalWritable := 'False'} : Bool;
            x24 { ExternalWritable := 'False'} : Bool;
            x25 { ExternalWritable := 'False'} : Bool;
            x26 { ExternalWritable := 'False'} : Bool;
            x27 { ExternalWritable := 'False'} : Bool;
            x28 { ExternalWritable := 'False'} : Bool;
            x29 { ExternalWritable := 'False'} : Bool;
            x30 { ExternalWritable := 'False'} : Bool;
            x31 { ExternalWritable := 'False'} : Bool;
         END_STRUCT;
      END_STRUCT;
      tHMR { ExternalWritable := 'False'} : Struct   // HMI Read
         xSpare0 { ExternalWritable := 'False'} : Bool;
         xSpare1 { ExternalWritable := 'False'} : Bool;
         xSpare2 { ExternalWritable := 'False'} : Bool;
         xSpare3 { ExternalWritable := 'False'} : Bool;
         xSpare4 { ExternalWritable := 'False'} : Bool;
         xSpare5 { ExternalWritable := 'False'} : Bool;
         xSpare6 { ExternalWritable := 'False'} : Bool;
         xSpare7 { ExternalWritable := 'False'} : Bool;
         xSpare8 { ExternalWritable := 'False'} : Bool;
         xSpare9 { ExternalWritable := 'False'} : Bool;
         xSpare10 { ExternalWritable := 'False'} : Bool;
         xSpare11 { ExternalWritable := 'False'} : Bool;
         xSpare12 { ExternalWritable := 'False'} : Bool;
         xSpare13 { ExternalWritable := 'False'} : Bool;
         xSpare14 { ExternalWritable := 'False'} : Bool;
         xSpare15 { ExternalWritable := 'False'} : Bool;
         xSpare16 { ExternalWritable := 'False'} : Bool;
         xSpare17 { ExternalWritable := 'False'} : Bool;
         xSpare18 { ExternalWritable := 'False'} : Bool;
         xSpare19 { ExternalWritable := 'False'} : Bool;
         xSpare20 { ExternalWritable := 'False'} : Bool;
         xSpare21 { ExternalWritable := 'False'} : Bool;
         xSpare22 { ExternalWritable := 'False'} : Bool;
         xSpare23 { ExternalWritable := 'False'} : Bool;
         xSpare24 { ExternalWritable := 'False'} : Bool;
         xSpare25 { ExternalWritable := 'False'} : Bool;
         xSpare26 { ExternalWritable := 'False'} : Bool;
         xSpare27 { ExternalWritable := 'False'} : Bool;
         xSpare28 { ExternalWritable := 'False'} : Bool;
         xSpare29 { ExternalWritable := 'False'} : Bool;
         xSpare30 { ExternalWritable := 'False'} : Bool;
         xSpare31 { ExternalWritable := 'False'} : Bool;
         xSpare { ExternalWritable := 'False'} : Array[0..15] of Bool;
         iSpare0 { ExternalWritable := 'False'} : Int;
         iSpare1 { ExternalWritable := 'False'} : Int;
         iSpare2 { ExternalWritable := 'False'} : Int;
         iSpare3 { ExternalWritable := 'False'} : Int;
         iSpare4 { ExternalWritable := 'False'} : Int;
         iSpare5 { ExternalWritable := 'False'} : Int;
         iSpare6 { ExternalWritable := 'False'} : Int;
         iSpare7 { ExternalWritable := 'False'} : Int;
         iSpare8 { ExternalWritable := 'False'} : Int;
         iSpare9 { ExternalWritable := 'False'} : Int;
         iSpare10 { ExternalWritable := 'False'} : Int;
         iSpare11 { ExternalWritable := 'False'} : Int;
         iSpare12 { ExternalWritable := 'False'} : Int;
         iSpare13 { ExternalWritable := 'False'} : Int;
         iSpare14 { ExternalWritable := 'False'} : Int;
         iSpare15 { ExternalWritable := 'False'} : Int;
         iSpare16 { ExternalWritable := 'False'} : Int;
         dHeadStatus_H1 { ExternalWritable := 'False'} : DInt;   // Head #1 firing status (1=OFF 3=ON) {x|x|x|x|O}
         dHeadStatus_H2 { ExternalWritable := 'False'} : DInt;   // Head #2 firing status (1=OFF 3=ON) {x|x|x|x|O}
         dHeadStatus_H3 { ExternalWritable := 'False'} : DInt;   // Head #3 firing status (1=OFF 3=ON) {x|x|x|x|O}
         dHeadStatus_H4 { ExternalWritable := 'False'} : DInt;   // Head #4 firing status (1=OFF 3=ON) {x|x|x|x|O}
         dHeadStatus_H5 { ExternalWritable := 'False'} : DInt;   // Head #5 firing status (1=OFF 3=ON) {x|x|x|x|O}
         dHeadStatus_H6 { ExternalWritable := 'False'} : DInt;   // Head #6 firing status (1=OFF 3=ON) {x|x|x|x|O}
         dHeadStatus_H7 { ExternalWritable := 'False'} : DInt;   // Head #7 firing status (1=OFF 3=ON) {x|x|x|x|O}
         dHeadStatus_H8 { ExternalWritable := 'False'} : DInt;   // Head #8 firing status (1=OFF 3=ON) {x|x|x|x|O}
         dSpare8 { ExternalWritable := 'False'} : DInt;
         dSpare9 { ExternalWritable := 'False'} : DInt;
         dSpare10 { ExternalWritable := 'False'} : DInt;
         dSpare11 { ExternalWritable := 'False'} : DInt;
         dSpare12 { ExternalWritable := 'False'} : DInt;
         dSpare13 { ExternalWritable := 'False'} : DInt;
         dSpare14 { ExternalWritable := 'False'} : DInt;
         dSpare15 { ExternalWritable := 'False'} : DInt;
         dSpare { ExternalWritable := 'False'} : Array[0..15] of DInt;
         rHeadUsage_km_H1 { ExternalWritable := 'False'} : Real;   // Head #1 head usage [km] {km|km|x|x|O}
         rHeadUsage_km_H2 { ExternalWritable := 'False'} : Real;   // Head #2 head usage [km] {km|km|x|x|O}
         rHeadUsage_km_H3 { ExternalWritable := 'False'} : Real;   // Head #3 head usage [km] {km|km|x|x|O}
         rHeadUsage_km_H4 { ExternalWritable := 'False'} : Real;   // Head #4 head usage [km] {km|km|x|x|O}
         rHeadUsage_km_H5 { ExternalWritable := 'False'} : Real;   // Head #5 head usage [km] {km|km|x|x|O}
         rHeadUsage_km_H6 { ExternalWritable := 'False'} : Real;   // Head #6 head usage [km] {km|km|x|x|O}
         rHeadUsage_km_H7 { ExternalWritable := 'False'} : Real;   // Head #7 head usage [km] {km|km|x|x|O}
         rHeadUsage_km_H8 { ExternalWritable := 'False'} : Real;   // Head #8 head usage [km] {km|km|x|x|O}
         rSpare8 { ExternalWritable := 'False'} : Real;
         tManCmd { ExternalWritable := 'False'} : Struct
            xMan_FireON_Fdbk_H1 { ExternalWritable := 'False'} : Bool;   // Head #1 manual fire ON Feeback {x|x|x|x|O}
            xMan_FireOFF_Fdbk_H1 { ExternalWritable := 'False'} : Bool;   // Head #1 manual fire OFF Feedback {x|x|x|x|O}
            xMan_OilON_Fdbk_H1 { ExternalWritable := 'False'} : Bool;   // Head #1 manual oil feedback ON {x|x|x|x|O}
            xMan_FireON_Fdbk_H2 { ExternalWritable := 'False'} : Bool;   // Head #2 manual fire ON Feeback {x|x|x|x|O}
            xMan_FireOFF_Fdbk_H2 { ExternalWritable := 'False'} : Bool;   // Head #2 manual fire OFF Feedback {x|x|x|x|O}
            xMan_OilON_Fdbk_H2 { ExternalWritable := 'False'} : Bool;   // Head #2 manual oil feedback ON {x|x|x|x|O}
            xMan_FireON_Fdbk_H3 { ExternalWritable := 'False'} : Bool;   // Head #3 manual fire ON Feeback {x|x|x|x|O}
            xMan_FireOFF_Fdbk_H3 { ExternalWritable := 'False'} : Bool;   // Head #3 manual fire OFF Feedback {x|x|x|x|O}
            xMan_OilON_Fdbk_H3 { ExternalWritable := 'False'} : Bool;   // Head #3 manual oil feedback ON {x|x|x|x|O}
            xMan_FireON_Fdbk_H4 { ExternalWritable := 'False'} : Bool;   // Head #4 manual fire ON Feeback {x|x|x|x|O}
            xMan_FireOFF_Fdbk_H4 { ExternalWritable := 'False'} : Bool;   // Head #4 manual fire OFF Feedback {x|x|x|x|O}
            xMan_OilON_Fdbk_H4 { ExternalWritable := 'False'} : Bool;   // Head #4 manual oil feedback ON {x|x|x|x|O}
            xMan_FireON_Fdbk_H5 { ExternalWritable := 'False'} : Bool;   // Head #5 manual fire ON Feeback {x|x|x|x|O}
            xMan_FireOFF_Fdbk_H5 { ExternalWritable := 'False'} : Bool;   // Head #5 manual fire OFF Feedback {x|x|x|x|O}
            xMan_OilON_Fdbk_H5 { ExternalWritable := 'False'} : Bool;   // Head #5 manual oil feedback ON {x|x|x|x|O}
            xMan_FireON_Fdbk_H6 { ExternalWritable := 'False'} : Bool;   // Head #6 manual fire ON Feeback {x|x|x|x|O}
            xMan_FireOFF_Fdbk_H6 { ExternalWritable := 'False'} : Bool;   // Head #6 manual fire OFF Feedback {x|x|x|x|O}
            xMan_OilON_Fdbk_H6 { ExternalWritable := 'False'} : Bool;   // Head #6 manual oil feedback ON {x|x|x|x|O}
            xMan_FireON_Fdbk_H7 { ExternalWritable := 'False'} : Bool;   // Head #7 manual fire ON Feeback {x|x|x|x|O}
            xMan_FireOFF_Fdbk_H7 { ExternalWritable := 'False'} : Bool;   // Head #7 manual fire OFF Feedback {x|x|x|x|O}
            xMan_OilON_Fdbk_H7 { ExternalWritable := 'False'} : Bool;   // Head #7 manual oil feedback ON {x|x|x|x|O}
            xMan_FireON_Fdbk_H8 { ExternalWritable := 'False'} : Bool;   // Head #8 manual fire ON Feeback {x|x|x|x|O}
            xMan_FireOFF_Fdbk_H8 { ExternalWritable := 'False'} : Bool;   // Head #8 manual fire OFF Feedback {x|x|x|x|O}
            xMan_OilON_Fdbk_H8 { ExternalWritable := 'False'} : Bool;   // Head #8 manual oil feedback ON {x|x|x|x|O}
            xSpare24 { ExternalWritable := 'False'} : Bool;
            xSpare25 { ExternalWritable := 'False'} : Bool;
            xSpare26 { ExternalWritable := 'False'} : Bool;
            xSpare27 { ExternalWritable := 'False'} : Bool;
            xSpare28 { ExternalWritable := 'False'} : Bool;
            xSpare29 { ExternalWritable := 'False'} : Bool;
            xSpare30 { ExternalWritable := 'False'} : Bool;
            xSpare31 { ExternalWritable := 'False'} : Bool;
         END_STRUCT;
      END_STRUCT;
      tHMW : Struct   // HMI Write
         xResetUsageCounter_H1 : Bool;   // Head #1 reset head usage counter {x|x|x|x|O}
         xResetUsageCounter_H2 : Bool;   // Head #2 reset head usage counter {x|x|x|x|O}
         xResetUsageCounter_H3 : Bool;   // Head #3 reset head usage counter {x|x|x|x|O}
         xResetUsageCounter_H4 : Bool;   // Head #4 reset head usage counter {x|x|x|x|O}
         xResetUsageCounter_H5 : Bool;   // Head #5 reset head usage counter {x|x|x|x|O}
         xResetUsageCounter_H6 : Bool;   // Head #6 reset head usage counter {x|x|x|x|O}
         xResetUsageCounter_H7 : Bool;   // Head #7 reset head usage counter {x|x|x|x|O}
         xResetUsageCounter_H8 : Bool;   // Head #8 reset head usage counter {x|x|x|x|O}
         xSpare8 : Bool;
         xSpare9 : Bool;
         xSpare10 : Bool;
         xSpare11 : Bool;
         xSpare12 : Bool;
         xSpare13 : Bool;
         xSpare14 : Bool;
         xSpare15 : Bool;
         xSpare16 : Bool;
         xSpare17 : Bool;
         xSpare18 : Bool;
         xSpare19 : Bool;
         xSpare20 : Bool;
         xSpare21 : Bool;
         xSpare22 : Bool;
         xSpare23 : Bool;
         xSpare24 : Bool;
         xSpare25 : Bool;
         xSpare26 : Bool;
         xSpare27 : Bool;
         xSpare28 : Bool;
         xSpare29 : Bool;
         xSpare30 : Bool;
         xSpare31 : Bool;
         xSpare : Array[0..15] of Bool;
         iSpare0 : Int;
         iSpare1 : Int;
         iSpare2 : Int;
         iSpare3 : Int;
         iSpare4 : Int;
         iSpare5 : Int;
         iSpare6 : Int;
         iSpare7 : Int;
         iSpare8 : Int;
         iSpare9 : Int;
         iSpare10 : Int;
         iSpare11 : Int;
         iSpare12 : Int;
         iSpare13 : Int;
         iSpare14 : Int;
         iSpare15 : Int;
         iSpare16 : Int;
         dHeadFireONReaction_ms_H1 : DInt;   // Head #1 fire ON reaction time [ms] {ms|s|0|1|M}
         dHeadFireOFFReaction_ms_H1 : DInt;   // Head #1 fire OFF reaction time [ms] {ms|s|0|1|M}
         dHeadOilONDelay_ms_H1 : DInt;   // Head #1 Oil ON delay [ms]{ms|s|-2|2|O}
         dHeadOilOFFDelay_ms_H1 : DInt;   // Head #1 Oil OFF delay [ms]{ms|s|-2|2|O}
         dHeadFireONDelay_cmm_H1 : DInt;   // Head #1 fire ON delay [mm/100] {mm/100|mm|-50|50|O}
         dHeadFireOFFDelay_cmm_H1 : DInt;   // Head #1 fire OFF delay [mm/100] {mm/100|mm|-50|50|O}
         dHeadPressure_mN_H1 : DInt;   // Head #1 pressure value [N/1000] {N/1000|N|16|180|O}
         dHeadFireONReaction_ms_H2 : DInt;   // Head #2 fire ON reaction time [ms] {ms|s|0|1|M}
         dHeadFireOFFReaction_ms_H2 : DInt;   // Head #2 fire OFF reaction time [ms] {ms|s|0|1|M}
         dHeadOilONDelay_ms_H2 : DInt;   // Head #2 Oil ON delay [ms]{ms|s|-2|2|O}
         dHeadOilOFFDelay_ms_H2 : DInt;   // Head #2 Oil OFF delay [ms]{ms|s|-2|2|O}
         dHeadFireONDelay_cmm_H2 : DInt;   // Head #2 fire ON delay [mm/100] {mm/100|mm|-50|50|O}
         dHeadFireOFFDelay_cmm_H2 : DInt;   // Head #2 fire OFF delay [mm/100] {mm/100|mm|-50|50|O}
         dHeadPressure_mN_H2 : DInt;   // Head #2 pressure value [N/1000] {N/1000|N|16|180|O}
         dHeadFireONReaction_ms_H3 : DInt;   // Head #3 fire ON reaction time [ms] {ms|s|0|1|M}
         dHeadFireOFFReaction_ms_H3 : DInt;   // Head #3 fire OFF reaction time [ms] {ms|s|0|1|M}
         dHeadOilONDelay_ms_H3 : DInt;   // Head #3 Oil ON delay [ms]{ms|s|-2|2|O}
         dHeadOilOFFDelay_ms_H3 : DInt;   // Head #3 Oil OFF delay [ms]{ms|s|-2|2|O}
         dHeadFireONDelay_cmm_H3 : DInt;   // Head #3 fire ON delay [mm/100] {mm/100|mm|-50|50|O}
         dHeadFireOFFDelay_cmm_H3 : DInt;   // Head #3 fire OFF delay [mm/100] {mm/100|mm|-50|50|O}
         dHeadPressure_mN_H3 : DInt;   // Head #3 pressure value [N/1000] {N/1000|N|16|180|O}
         dHeadFireONReaction_ms_H4 : DInt;   // Head #4 fire ON reaction time [ms] {ms|s|0|1|M}
         dHeadFireOFFReaction_ms_H4 : DInt;   // Head #4 fire OFF reaction time [ms] {ms|s|0|1|M}
         dHeadOilONDelay_ms_H4 : DInt;   // Head #4 Oil ON delay [ms]{ms|s|-2|2|O}
         dHeadOilOFFDelay_ms_H4 : DInt;   // Head #4 Oil OFF delay [ms]{ms|s|-2|2|O}
         dHeadFireONDelay_cmm_H4 : DInt;   // Head #4 fire ON delay [mm/100] {mm/100|mm|-50|50|O}
         dHeadFireOFFDelay_cmm_H4 : DInt;   // Head #4 fire OFF delay [mm/100] {mm/100|mm|-50|50|O}
         dHeadPressure_mN_H4 : DInt;   // Head #4 pressure value [N/1000] {N/1000|N|16|180|O}
         dHeadFireONReaction_ms_H5 : DInt;   // Head #5 fire ON reaction time [ms] {ms|s|0|1|M}
         dHeadFireOFFReaction_ms_H5 : DInt;   // Head #5 fire OFF reaction time [ms] {ms|s|0|1|M}
         dHeadOilONDelay_ms_H5 : DInt;   // Head #5 Oil ON delay [ms]{ms|s|-2|2|O}
         dHeadOilOFFDelay_ms_H5 : DInt;   // Head #5 Oil OFF delay [ms]{ms|s|-2|2|O}
         dHeadFireONDelay_cmm_H5 : DInt;   // Head #5 fire ON delay [mm/100] {mm/100|mm|-50|50|O}
         dHeadFireOFFDelay_cmm_H5 : DInt;   // Head #5 fire OFF delay [mm/100] {mm/100|mm|-50|50|O}
         dHeadPressure_mN_H5 : DInt;   // Head #5 pressure value [N/1000] {N/1000|N|16|180|O}
         dHeadFireONReaction_ms_H6 : DInt;   // Head #6 fire ON reaction time [ms] {ms|s|0|1|M}
         dHeadFireOFFReaction_ms_H6 : DInt;   // Head #6 fire OFF reaction time [ms] {ms|s|0|1|M}
         dHeadOilONDelay_ms_H6 : DInt;   // Head #6 Oil ON delay [ms]{ms|s|-2|2|O}
         dHeadOilOFFDelay_ms_H6 : DInt;   // Head #6 Oil OFF delay [ms]{ms|s|-2|2|O}
         dHeadFireONDelay_cmm_H6 : DInt;   // Head #6 fire ON delay [mm/100] {mm/100|mm|-50|50|O}
         dHeadFireOFFDelay_cmm_H6 : DInt;   // Head #6 fire OFF delay [mm/100] {mm/100|mm|-50|50|O}
         dHeadPressure_mN_H6 : DInt;   // Head #6 pressure value [N/1000] {N/1000|N|16|180|O}
         dHeadFireONReaction_ms_H7 : DInt;   // Head #7 fire ON reaction time [ms] {ms|s|0|1|M}
         dHeadFireOFFReaction_ms_H7 : DInt;   // Head #7 fire OFF reaction time [ms] {ms|s|0|1|M}
         dHeadOilONDelay_ms_H7 : DInt;   // Head #7 Oil ON delay [ms]{ms|s|-2|2|O}
         dHeadOilOFFDelay_ms_H7 : DInt;   // Head #7 Oil OFF delay [ms]{ms|s|-2|2|O}
         dHeadFireONDelay_cmm_H7 : DInt;   // Head #7 fire ON delay [mm/100] {mm/100|mm|-50|50|O}
         dHeadFireOFFDelay_cmm_H7 : DInt;   // Head #7 fire OFF delay [mm/100] {mm/100|mm|-50|50|O}
         dHeadPressure_mN_H7 : DInt;   // Head #7 pressure value [N/1000] {N/1000|N|16|180|O}
         dHeadFireONReaction_ms_H8 : DInt;   // Head #8 fire ON reaction time [ms] {ms|s|0|1|M}
         dHeadFireOFFReaction_ms_H8 : DInt;   // Head #8 fire OFF reaction time [ms] {ms|s|0|1|M}
         dHeadOilONDelay_ms_H8 : DInt;   // Head #8 Oil ON delay [ms]{ms|s|-2|2|O}
         dHeadOilOFFDelay_ms_H8 : DInt;   // Head #8 Oil OFF delay [ms]{ms|s|-2|2|O}
         dHeadFireONDelay_cmm_H8 : DInt;   // Head #8 fire ON delay [mm/100] {mm/100|mm|-50|50|O}
         dHeadFireOFFDelay_cmm_H8 : DInt;   // Head #8 fire OFF delay [mm/100] {mm/100|mm|-50|50|O}
         dHeadPressure_mN_H8 : DInt;   // Head #8 pressure value [N/1000] {N/1000|N|16|180|O}
         dSpare56 : DInt;
         dSpare57 : DInt;
         dSpare58 : DInt;
         dSpare59 : DInt;
         rSpare0 : Real;
         rSpare1 : Real;
         rSpare2 : Real;
         rSpare3 : Real;
         rSpare4 : Real;
         rSpare5 : Real;
         rSpare6 : Real;
         rSpare7 : Real;
         rSpare8 : Real;
         tManCmd : Struct
            xMan_FireON_H1 : Bool;   // Head #1 manual fire ON {x|x|x|x|O}
            xMan_FireOFF_H1 : Bool;   // Head #1 manual fire OFF {x|x|x|x|O}
            xMan_OilON_H1 : Bool;   // Head #1 manual oil ON {x|x|x|x|O}
            xMan_FireON_H2 : Bool;   // Head #2 manual fire ON {x|x|x|x|O}
            xMan_FireOFF_H2 : Bool;   // Head #2 manual fire OFF {x|x|x|x|O}
            xMan_OilON_H2 : Bool;   // Head #2 manual oil ON {x|x|x|x|O}
            xMan_FireON_H3 : Bool;   // Head #3 manual fire ON {x|x|x|x|O}
            xMan_FireOFF_H3 : Bool;   // Head #3 manual fire OFF {x|x|x|x|O}
            xMan_OilON_H3 : Bool;   // Head #3 manual oil ON {x|x|x|x|O}
            xMan_FireON_H4 : Bool;   // Head #4 manual fire ON {x|x|x|x|O}
            xMan_FireOFF_H4 : Bool;   // Head #4 manual fire OFF {x|x|x|x|O}
            xMan_OilON_H4 : Bool;   // Head #4 manual oil ON {x|x|x|x|O}
            xMan_FireON_H5 : Bool;   // Head #5 manual fire ON {x|x|x|x|O}
            xMan_FireOFF_H5 : Bool;   // Head #5 manual fire OFF {x|x|x|x|O}
            xMan_OilON_H5 : Bool;   // Head #5 manual oil ON {x|x|x|x|O}
            xMan_FireON_H6 : Bool;   // Head #6 manual fire ON {x|x|x|x|O}
            xMan_FireOFF_H6 : Bool;   // Head #6 manual fire OFF {x|x|x|x|O}
            xMan_OilON_H6 : Bool;   // Head #6 manual oil ON {x|x|x|x|O}
            xMan_FireON_H7 : Bool;   // Head #7 manual fire ON {x|x|x|x|O}
            xMan_FireOFF_H7 : Bool;   // Head #7 manual fire OFF {x|x|x|x|O}
            xMan_OilON_H7 : Bool;   // Head #7 manual oil ON {x|x|x|x|O}
            xMan_FireON_H8 : Bool;   // Head #8 manual fire ON {x|x|x|x|O}
            xMan_FireOFF_H8 : Bool;   // Head #8 manual fire OFF {x|x|x|x|O}
            xMan_OilON_H8 : Bool;   // Head #8 manual oil ON {x|x|x|x|O}
            xSpare24 : Bool;
            xSpare25 : Bool;
            xSpare26 : Bool;
            xSpare27 : Bool;
            xSpare28 : Bool;
            xSpare29 : Bool;
            xSpare30 : Bool;
            xSpare31 : Bool;
         END_STRUCT;
      END_STRUCT;
   END_STRUCT;


BEGIN
   tHMR.xSpare15 := FALSE;
   tHMR.dSpare8 := 0;
   tHMR.dSpare9 := 0;
   tHMR.dSpare10 := 0;
   tHMR.dSpare11 := 0;
   tHMW.xResetUsageCounter_H2 := FALSE;
   tHMW.xResetUsageCounter_H3 := FALSE;
   tHMW.xResetUsageCounter_H4 := FALSE;
   tHMW.xResetUsageCounter_H5 := FALSE;
   tHMW.xResetUsageCounter_H6 := FALSE;
   tHMW.xResetUsageCounter_H7 := FALSE;
   tHMW.xResetUsageCounter_H8 := FALSE;
   tHMW.xSpare8 := FALSE;
   tHMW.xSpare14 := FALSE;
   tHMW.xSpare15 := FALSE;
   tHMW.xSpare16 := TRUE;
   tHMW.xSpare17 := TRUE;
   tHMW.xSpare18 := TRUE;
   tHMW.xSpare19 := TRUE;
   tHMW.xSpare20 := TRUE;
   tHMW.xSpare21 := TRUE;
   tHMW.xSpare22 := TRUE;
   tHMW.xSpare23 := TRUE;
   tHMW.iSpare16 := 0;

END_DATA_BLOCK

DATA_BLOCK "DB_M256M_Scada"
{ DB_Accessible_From_OPC_UA := 'FALSE' ;
 DB_Accessible_From_Webserver := 'FALSE' ;
 S7_Optimized_Access := 'FALSE' }
VERSION : 0.1
NON_RETAIN
   STRUCT
      tAlm : Struct   // HMI Alarms
         tE { ExternalWritable := 'False'} : Struct
            x0 { ExternalWritable := 'False'} : Bool;
            x1 { ExternalWritable := 'False'} : Bool;
            x2 { ExternalWritable := 'False'} : Bool;
            x3 { ExternalWritable := 'False'} : Bool;
            x4 { ExternalWritable := 'False'} : Bool;
            x5 { ExternalWritable := 'False'} : Bool;
            x6 { ExternalWritable := 'False'} : Bool;
            x7 { ExternalWritable := 'False'} : Bool;
            x8 { ExternalWritable := 'False'} : Bool;
            x9 { ExternalWritable := 'False'} : Bool;
            x10 { ExternalWritable := 'False'} : Bool;
            x11 { ExternalWritable := 'False'} : Bool;
            x12 { ExternalWritable := 'False'} : Bool;
            x13 { ExternalWritable := 'False'} : Bool;
            x14 { ExternalWritable := 'False'} : Bool;
            x15 { ExternalWritable := 'False'} : Bool;
            x16 { ExternalWritable := 'False'} : Bool;
            x17 { ExternalWritable := 'False'} : Bool;
            x18 { ExternalWritable := 'False'} : Bool;
            x19 { ExternalWritable := 'False'} : Bool;
            x20 { ExternalWritable := 'False'} : Bool;
            x21 { ExternalWritable := 'False'} : Bool;
            x22 { ExternalWritable := 'False'} : Bool;
            x23 { ExternalWritable := 'False'} : Bool;
            x24 { ExternalWritable := 'False'} : Bool;
            x25 { ExternalWritable := 'False'} : Bool;
            x26 { ExternalWritable := 'False'} : Bool;
            x27 { ExternalWritable := 'False'} : Bool;
            x28 { ExternalWritable := 'False'} : Bool;
            x29 { ExternalWritable := 'False'} : Bool;
            x30 { ExternalWritable := 'False'} : Bool;
            x31 { ExternalWritable := 'False'} : Bool;
         END_STRUCT;
         tS { ExternalWritable := 'False'} : Struct
            tS0 { ExternalWritable := 'False'} : Struct
               x0 { ExternalWritable := 'False'} : Bool;   // Head#1.Initialization timeout
               x1 { ExternalWritable := 'False'} : Bool;   // Head#1.homing timeout
               x2 { ExternalWritable := 'False'} : Bool;   // Head#1.positioning timeout
               x3 { ExternalWritable := 'False'} : Bool;   // Head#1.carriage overload
               x4 { ExternalWritable := 'False'} : Bool;   // Head#1.drive error
               x5 { ExternalWritable := 'False'} : Bool;   // Head#1.missing ethernet IP connection
               x6 { ExternalWritable := 'False'} : Bool;   // Head#1.op.side overstroke
               x7 { ExternalWritable := 'False'} : Bool;   // Head#1.oppo.op.side overstroke
               x8 { ExternalWritable := 'False'} : Bool;   // Head#1.overstroke
               x9 { ExternalWritable := 'False'} : Bool;   // Head#2.Initialization timeout
               x10 { ExternalWritable := 'False'} : Bool;   // Head#2.homing timeout
               x11 { ExternalWritable := 'False'} : Bool;   // Head#2.positioning timeout
               x12 { ExternalWritable := 'False'} : Bool;   // Head#2.carriage overload
               x13 { ExternalWritable := 'False'} : Bool;   // Head#2.drive error
               x14 { ExternalWritable := 'False'} : Bool;   // Head#2.missing ethernet IP connection
               x15 { ExternalWritable := 'False'} : Bool;   // Head#2.op.side overstroke
               x16 { ExternalWritable := 'False'} : Bool;   // Head#2.oppo.op.side overstroke
               x17 { ExternalWritable := 'False'} : Bool;   // Head#2.overstroke
               x18 { ExternalWritable := 'False'} : Bool;   // Head#3.Initialization timeout
               x19 { ExternalWritable := 'False'} : Bool;   // Head#3.homing timeout
               x20 { ExternalWritable := 'False'} : Bool;   // Head#3.positioning timeout
               x21 { ExternalWritable := 'False'} : Bool;   // Head#3.carriage overload
               x22 { ExternalWritable := 'False'} : Bool;   // Head#3.drive error
               x23 { ExternalWritable := 'False'} : Bool;   // Head#3.missing ethernet IP connection
               x24 { ExternalWritable := 'False'} : Bool;   // Head#3.op.side overstroke
               x25 { ExternalWritable := 'False'} : Bool;   // Head#3.oppo.op.side overstroke
               x26 { ExternalWritable := 'False'} : Bool;   // Head#3.overstroke
               x27 { ExternalWritable := 'False'} : Bool;
               x28 { ExternalWritable := 'False'} : Bool;
               x29 { ExternalWritable := 'False'} : Bool;
               x30 { ExternalWritable := 'False'} : Bool;
               x31 { ExternalWritable := 'False'} : Bool;
            END_STRUCT;
            tS1 { ExternalWritable := 'False'} : Struct
               x0 { ExternalWritable := 'False'} : Bool;   // Head#4.Initialization timeout
               x1 { ExternalWritable := 'False'} : Bool;   // Head#4.homing timeout
               x2 { ExternalWritable := 'False'} : Bool;   // Head#4.positioning timeout
               x3 { ExternalWritable := 'False'} : Bool;   // Head#4.carriage overload
               x4 { ExternalWritable := 'False'} : Bool;   // Head#4.drive error
               x5 { ExternalWritable := 'False'} : Bool;   // Head#4.missing ethernet IP connection
               x6 { ExternalWritable := 'False'} : Bool;   // Head#4.op.side overstroke
               x7 { ExternalWritable := 'False'} : Bool;   // Head#4.oppo.op.side overstroke
               x8 { ExternalWritable := 'False'} : Bool;   // Head#4.overstroke
               x9 { ExternalWritable := 'False'} : Bool;   // Head#5.Initialization timeout
               x10 { ExternalWritable := 'False'} : Bool;   // Head#5.homing timeout
               x11 { ExternalWritable := 'False'} : Bool;   // Head#5.positioning timeout
               x12 { ExternalWritable := 'False'} : Bool;   // Head#5.carriage overload
               x13 { ExternalWritable := 'False'} : Bool;   // Head#5.drive error
               x14 { ExternalWritable := 'False'} : Bool;   // Head#5.missing ethernet IP connection
               x15 { ExternalWritable := 'False'} : Bool;   // Head#5.op.side overstroke
               x16 { ExternalWritable := 'False'} : Bool;   // Head#5.oppo.op.side overstroke
               x17 { ExternalWritable := 'False'} : Bool;   // Head#5.overstroke
               x18 { ExternalWritable := 'False'} : Bool;   // Head#6.Initialization timeout
               x19 { ExternalWritable := 'False'} : Bool;   // Head#6.homing timeout
               x20 { ExternalWritable := 'False'} : Bool;   // Head#6.positioning timeout
               x21 { ExternalWritable := 'False'} : Bool;   // Head#6.carriage overload
               x22 { ExternalWritable := 'False'} : Bool;   // Head#6.drive error
               x23 { ExternalWritable := 'False'} : Bool;   // Head#6.missing ethernet IP connection
               x24 { ExternalWritable := 'False'} : Bool;   // Head#6.op.side overstroke
               x25 { ExternalWritable := 'False'} : Bool;   // Head#6.oppo.op.side overstroke
               x26 { ExternalWritable := 'False'} : Bool;   // Head#6.overstroke
               x27 { ExternalWritable := 'False'} : Bool;
               x28 { ExternalWritable := 'False'} : Bool;
               x29 { ExternalWritable := 'False'} : Bool;
               x30 { ExternalWritable := 'False'} : Bool;
               x31 { ExternalWritable := 'False'} : Bool;
            END_STRUCT;
            tS2 { ExternalWritable := 'False'} : Struct
               x0 { ExternalWritable := 'False'} : Bool;   // Head#7.Initialization timeout
               x1 { ExternalWritable := 'False'} : Bool;   // Head#7.homing timeout
               x2 { ExternalWritable := 'False'} : Bool;   // Head#7.positioning timeout
               x3 { ExternalWritable := 'False'} : Bool;   // Head#7.carriage overload
               x4 { ExternalWritable := 'False'} : Bool;   // Head#7.drive error
               x5 { ExternalWritable := 'False'} : Bool;   // Head#7.missing ethernet IP connection
               x6 { ExternalWritable := 'False'} : Bool;   // Head#7.op.side overstroke
               x7 { ExternalWritable := 'False'} : Bool;   // Head#7.oppo.op.side overstroke
               x8 { ExternalWritable := 'False'} : Bool;   // Head#7.overstroke
               x9 { ExternalWritable := 'False'} : Bool;   // Head#8.Initialization timeout
               x10 { ExternalWritable := 'False'} : Bool;   // Head#8.homing timeout
               x11 { ExternalWritable := 'False'} : Bool;   // Head#8.positioning timeout
               x12 { ExternalWritable := 'False'} : Bool;   // Head#8.carriage overload
               x13 { ExternalWritable := 'False'} : Bool;   // Head#8.drive error
               x14 { ExternalWritable := 'False'} : Bool;   // Head#8.missing ethernet IP connection
               x15 { ExternalWritable := 'False'} : Bool;   // Head#8.op.side overstroke
               x16 { ExternalWritable := 'False'} : Bool;   // Head#8.oppo.op.side overstroke
               x17 { ExternalWritable := 'False'} : Bool;   // Head#8.overstroke
               x18 { ExternalWritable := 'False'} : Bool;
               x19 { ExternalWritable := 'False'} : Bool;
               x20 { ExternalWritable := 'False'} : Bool;
               x21 { ExternalWritable := 'False'} : Bool;
               x22 { ExternalWritable := 'False'} : Bool;
               x23 { ExternalWritable := 'False'} : Bool;
               x24 { ExternalWritable := 'False'} : Bool;
               x25 { ExternalWritable := 'False'} : Bool;
               x26 { ExternalWritable := 'False'} : Bool;
               x27 { ExternalWritable := 'False'} : Bool;
               x28 { ExternalWritable := 'False'} : Bool;
               x29 { ExternalWritable := 'False'} : Bool;
               x30 { ExternalWritable := 'False'} : Bool;
               x31 { ExternalWritable := 'False'} : Bool;
            END_STRUCT;
            tS3 { ExternalWritable := 'False'} : Struct
               x0 { ExternalWritable := 'False'} : Bool;
               x1 { ExternalWritable := 'False'} : Bool;
               x2 { ExternalWritable := 'False'} : Bool;
               x3 { ExternalWritable := 'False'} : Bool;
               x4 { ExternalWritable := 'False'} : Bool;
               x5 { ExternalWritable := 'False'} : Bool;
               x6 { ExternalWritable := 'False'} : Bool;
               x7 { ExternalWritable := 'False'} : Bool;
               x8 { ExternalWritable := 'False'} : Bool;
               x9 { ExternalWritable := 'False'} : Bool;
               x10 { ExternalWritable := 'False'} : Bool;
               x11 { ExternalWritable := 'False'} : Bool;
               x12 { ExternalWritable := 'False'} : Bool;
               x13 { ExternalWritable := 'False'} : Bool;
               x14 { ExternalWritable := 'False'} : Bool;
               x15 { ExternalWritable := 'False'} : Bool;
               x16 { ExternalWritable := 'False'} : Bool;
               x17 { ExternalWritable := 'False'} : Bool;
               x18 { ExternalWritable := 'False'} : Bool;
               x19 { ExternalWritable := 'False'} : Bool;
               x20 { ExternalWritable := 'False'} : Bool;
               x21 { ExternalWritable := 'False'} : Bool;
               x22 { ExternalWritable := 'False'} : Bool;
               x23 { ExternalWritable := 'False'} : Bool;
               x24 { ExternalWritable := 'False'} : Bool;
               x25 { ExternalWritable := 'False'} : Bool;
               x26 { ExternalWritable := 'False'} : Bool;
               x27 { ExternalWritable := 'False'} : Bool;
               x28 { ExternalWritable := 'False'} : Bool;
               x29 { ExternalWritable := 'False'} : Bool;
               x30 { ExternalWritable := 'False'} : Bool;
               x31 { ExternalWritable := 'False'} : Bool;
            END_STRUCT;
         END_STRUCT;
         tF { ExternalWritable := 'False'} : Struct
            x0 { ExternalWritable := 'False'} : Bool;
            x1 { ExternalWritable := 'False'} : Bool;
            x2 { ExternalWritable := 'False'} : Bool;
            x3 { ExternalWritable := 'False'} : Bool;
            x4 { ExternalWritable := 'False'} : Bool;
            x5 { ExternalWritable := 'False'} : Bool;
            x6 { ExternalWritable := 'False'} : Bool;
            x7 { ExternalWritable := 'False'} : Bool;
            x8 { ExternalWritable := 'False'} : Bool;
            x9 { ExternalWritable := 'False'} : Bool;
            x10 { ExternalWritable := 'False'} : Bool;
            x11 { ExternalWritable := 'False'} : Bool;
            x12 { ExternalWritable := 'False'} : Bool;
            x13 { ExternalWritable := 'False'} : Bool;
            x14 { ExternalWritable := 'False'} : Bool;
            x15 { ExternalWritable := 'False'} : Bool;
            x16 { ExternalWritable := 'False'} : Bool;
            x17 { ExternalWritable := 'False'} : Bool;
            x18 { ExternalWritable := 'False'} : Bool;
            x19 { ExternalWritable := 'False'} : Bool;
            x20 { ExternalWritable := 'False'} : Bool;
            x21 { ExternalWritable := 'False'} : Bool;
            x22 { ExternalWritable := 'False'} : Bool;
            x23 { ExternalWritable := 'False'} : Bool;
            x24 { ExternalWritable := 'False'} : Bool;
            x25 { ExternalWritable := 'False'} : Bool;
            x26 { ExternalWritable := 'False'} : Bool;
            x27 { ExternalWritable := 'False'} : Bool;
            x28 { ExternalWritable := 'False'} : Bool;
            x29 { ExternalWritable := 'False'} : Bool;
            x30 { ExternalWritable := 'False'} : Bool;
            x31 { ExternalWritable := 'False'} : Bool;
         END_STRUCT;
         tW { ExternalWritable := 'False'} : Struct
            x0 { ExternalWritable := 'False'} : Bool;
            x1 { ExternalWritable := 'False'} : Bool;
            x2 { ExternalWritable := 'False'} : Bool;
            x3 { ExternalWritable := 'False'} : Bool;
            x4 { ExternalWritable := 'False'} : Bool;
            x5 { ExternalWritable := 'False'} : Bool;
            x6 { ExternalWritable := 'False'} : Bool;
            x7 { ExternalWritable := 'False'} : Bool;
            x8 { ExternalWritable := 'False'} : Bool;
            x9 { ExternalWritable := 'False'} : Bool;
            x10 { ExternalWritable := 'False'} : Bool;
            x11 { ExternalWritable := 'False'} : Bool;
            x12 { ExternalWritable := 'False'} : Bool;
            x13 { ExternalWritable := 'False'} : Bool;
            x14 { ExternalWritable := 'False'} : Bool;
            x15 { ExternalWritable := 'False'} : Bool;
            x16 { ExternalWritable := 'False'} : Bool;
            x17 { ExternalWritable := 'False'} : Bool;
            x18 { ExternalWritable := 'False'} : Bool;
            x19 { ExternalWritable := 'False'} : Bool;
            x20 { ExternalWritable := 'False'} : Bool;
            x21 { ExternalWritable := 'False'} : Bool;
            x22 { ExternalWritable := 'False'} : Bool;
            x23 { ExternalWritable := 'False'} : Bool;
            x24 { ExternalWritable := 'False'} : Bool;
            x25 { ExternalWritable := 'False'} : Bool;
            x26 { ExternalWritable := 'False'} : Bool;
            x27 { ExternalWritable := 'False'} : Bool;
            x28 { ExternalWritable := 'False'} : Bool;
            x29 { ExternalWritable := 'False'} : Bool;
            x30 { ExternalWritable := 'False'} : Bool;
            x31 { ExternalWritable := 'False'} : Bool;
         END_STRUCT;
      END_STRUCT;
      tHMR { ExternalWritable := 'False'} : Struct   // HMI Read
         xSpare0 { ExternalWritable := 'False'} : Bool;   //
         xSpare1 { ExternalWritable := 'False'} : Bool;
         xSpare2 { ExternalWritable := 'False'} : Bool;
         xSpare3 { ExternalWritable := 'False'} : Bool;
         xSpare4 { ExternalWritable := 'False'} : Bool;
         xSpare5 { ExternalWritable := 'False'} : Bool;
         xSpare6 { ExternalWritable := 'False'} : Bool;
         xSpare7 { ExternalWritable := 'False'} : Bool;
         xSpare8 { ExternalWritable := 'False'} : Bool;
         xSpare9 { ExternalWritable := 'False'} : Bool;
         xSpare10 { ExternalWritable := 'False'} : Bool;
         xSpare11 { ExternalWritable := 'False'} : Bool;
         xSpare12 { ExternalWritable := 'False'} : Bool;
         xSpare13 { ExternalWritable := 'False'} : Bool;
         xSpare14 { ExternalWritable := 'False'} : Bool;
         xSpare15 { ExternalWritable := 'False'} : Bool;
         xSpare16 { ExternalWritable := 'False'} : Bool;
         xSpare17 { ExternalWritable := 'False'} : Bool;
         xSpare18 { ExternalWritable := 'False'} : Bool;
         xSpare19 { ExternalWritable := 'False'} : Bool;
         xSpare20 { ExternalWritable := 'False'} : Bool;
         xSpare21 { ExternalWritable := 'False'} : Bool;
         xSpare22 { ExternalWritable := 'False'} : Bool;
         xSpare23 { ExternalWritable := 'False'} : Bool;
         xSpare24 { ExternalWritable := 'False'} : Bool;
         xSpare25 { ExternalWritable := 'False'} : Bool;
         xSpare26 { ExternalWritable := 'False'} : Bool;
         xSpare27 { ExternalWritable := 'False'} : Bool;
         xSpare28 { ExternalWritable := 'False'} : Bool;
         xSpare29 { ExternalWritable := 'False'} : Bool;
         xSpare30 { ExternalWritable := 'False'} : Bool;
         xSpare31 { ExternalWritable := 'False'} : Bool;
         xSpare { ExternalWritable := 'False'} : Array[0..15] of Bool;
         iCodeAlarm_H1 { ExternalWritable := 'False'} : Int;   // Motor error code H1
         iCodeAlarm_H2 { ExternalWritable := 'False'} : Int;   // Motor error code H2
         iCodeAlarm_H3 { ExternalWritable := 'False'} : Int;   // Motor error code H3
         iCodeAlarm_H4 { ExternalWritable := 'False'} : Int;   // Motor error code H4
         iCodeAlarm_H5 { ExternalWritable := 'False'} : Int;   // Motor error code H5
         iCodeAlarm_H6 { ExternalWritable := 'False'} : Int;   // Motor error code H6
         iCodeAlarm_H7 { ExternalWritable := 'False'} : Int;   // Motor error code H7
         iCodeAlarm_H8 { ExternalWritable := 'False'} : Int;   // Motor error code H8
         iSpare8 { ExternalWritable := 'False'} : Int;
         iSpare9 { ExternalWritable := 'False'} : Int;
         iSpare10 { ExternalWritable := 'False'} : Int;
         iSpare11 { ExternalWritable := 'False'} : Int;
         iSpare12 { ExternalWritable := 'False'} : Int;
         iSpare13 { ExternalWritable := 'False'} : Int;
         iSpare14 { ExternalWritable := 'False'} : Int;
         iSpare15 { ExternalWritable := 'False'} : Int;
         iSpare16 { ExternalWritable := 'False'} : Int;
         dHeadActualPositions_cmm_H1 { ExternalWritable := 'False'} : DInt;   // Head#1 head actual position [mm/100] {mm/100|mm|x|x|O}
         dHeadActualPositions_cmm_H2 { ExternalWritable := 'False'} : DInt;   // Head#2 head actual position [mm/100] {mm/100|mm|x|x|O}
         dHeadActualPositions_cmm_H3 { ExternalWritable := 'False'} : DInt;   // Head#3 head actual position [mm/100] {mm/100|mm|x|x|O}
         dHeadActualPositions_cmm_H4 { ExternalWritable := 'False'} : DInt;   // Head#4 head actual position [mm/100] {mm/100|mm|x|x|O}
         dHeadActualPositions_cmm_H5 { ExternalWritable := 'False'} : DInt;   // Head#5 head actual position [mm/100] {mm/100|mm|x|x|O}
         dHeadActualPositions_cmm_H6 { ExternalWritable := 'False'} : DInt;   // Head#6 head actual position [mm/100] {mm/100|mm|x|x|O}
         dHeadActualPositions_cmm_H7 { ExternalWritable := 'False'} : DInt;   // Head#7 head actual position [mm/100] {mm/100|mm|x|x|O}
         dHeadActualPositions_cmm_H8 { ExternalWritable := 'False'} : DInt;   // Head#8 head actual position [mm/100] {mm/100|mm|x|x|O}
         dHeadHomePositions_cmm_H1 { ExternalWritable := 'False'} : DInt;   // Head#1 home position [mm/100] {mm/100|mm|x|x|O}
         dHeadHomePositions_cmm_H2 { ExternalWritable := 'False'} : DInt;   // Head#2 home position [mm/100] {mm/100|mm|x|x|O}
         dHeadHomePositions_cmm_H3 { ExternalWritable := 'False'} : DInt;   // Head#3 home position [mm/100] {mm/100|mm|x|x|O}
         dHeadHomePositions_cmm_H4 { ExternalWritable := 'False'} : DInt;   // Head#4 home position [mm/100] {mm/100|mm|x|x|O}
         dHeadHomePositions_cmm_H5 { ExternalWritable := 'False'} : DInt;   // Head#5 home position [mm/100] {mm/100|mm|x|x|O}
         dHeadHomePositions_cmm_H6 { ExternalWritable := 'False'} : DInt;   // Head#6 home position [mm/100] {mm/100|mm|x|x|O}
         dHeadHomePositions_cmm_H7 { ExternalWritable := 'False'} : DInt;   // Head#7 home position [mm/100] {mm/100|mm|x|x|O}
         dHeadHomePositions_cmm_H8 { ExternalWritable := 'False'} : DInt;   // Head#8 home position [mm/100] {mm/100|mm|x|x|O}
         dHeadMoveStatus_H1 { ExternalWritable := 'False'} : DInt;   // Head#1 move status (1=Not Initialized 2=Not referred 3=Not positioned 4=Positioned 5=Positioning 6=Virtual collision 7=Anomaly) {x|x|x|x|O}
         dHeadMoveStatus_H2 { ExternalWritable := 'False'} : DInt;   // Head#2 move status (1=Not Initialized 2=Not referred 3=Not positioned 4=Positioned 5=Positioning 6=Virtual collision 7=Anomaly) {x|x|x|x|O}
         dHeadMoveStatus_H3 { ExternalWritable := 'False'} : DInt;   // Head#3 move status (1=Not Initialized 2=Not referred 3=Not positioned 4=Positioned 5=Positioning 6=Virtual collision 7=Anomaly) {x|x|x|x|O}
         dHeadMoveStatus_H4 { ExternalWritable := 'False'} : DInt;   // Head#4 move status (1=Not Initialized 2=Not referred 3=Not positioned 4=Positioned 5=Positioning 6=Virtual collision 7=Anomaly) {x|x|x|x|O}
         dHeadMoveStatus_H5 { ExternalWritable := 'False'} : DInt;   // Head#5 move status (1=Not Initialized 2=Not referred 3=Not positioned 4=Positioned 5=Positioning 6=Virtual collision 7=Anomaly) {x|x|x|x|O}
         dHeadMoveStatus_H6 { ExternalWritable := 'False'} : DInt;   // Head#6 move status (1=Not Initialized 2=Not referred 3=Not positioned 4=Positioned 5=Positioning 6=Virtual collision 7=Anomaly) {x|x|x|x|O}
         dHeadMoveStatus_H7 { ExternalWritable := 'False'} : DInt;   // Head#7 move status (1=Not Initialized 2=Not referred 3=Not positioned 4=Positioned 5=Positioning 6=Virtual collision 7=Anomaly) {x|x|x|x|O}
         dHeadMoveStatus_H8 { ExternalWritable := 'False'} : DInt;   // Head#8 move status (1=Not Initialized 2=Not referred 3=Not positioned 4=Positioned 5=Positioning 6=Virtual collision 7=Anomaly) {x|x|x|x|O}
         dSpare { ExternalWritable := 'False'} : Array[0..7] of DInt;
         rSpare0 { ExternalWritable := 'False'} : Real;
         rSpare1 { ExternalWritable := 'False'} : Real;
         rSpare2 { ExternalWritable := 'False'} : Real;
         rSpare3 { ExternalWritable := 'False'} : Real;
         rSpare4 { ExternalWritable := 'False'} : Real;
         rSpare5 { ExternalWritable := 'False'} : Real;
         rSpare6 { ExternalWritable := 'False'} : Real;
         rSpare7 { ExternalWritable := 'False'} : Real;
         rSpare8 { ExternalWritable := 'False'} : Real;
         tManCmd { ExternalWritable := 'False'} : Struct
            xManJogForwardFdbk_H1 { ExternalWritable := 'False'} : Bool;   // Head#1 manual jog forward fdbk {x|x|x|x|O}
            xManJogBackwardFdbk_H1 { ExternalWritable := 'False'} : Bool;   // Head#1 manual jog backward fdbk {x|x|x|x|O}
            xManJogForwardFdbk_H2 { ExternalWritable := 'False'} : Bool;   // Head#2 manual jog forward fdbk {x|x|x|x|O}
            xManJogBackwardFdbk_H2 { ExternalWritable := 'False'} : Bool;   // Head#2 manual jog backward fdbk {x|x|x|x|O}
            xManJogForwardFdbk_H3 { ExternalWritable := 'False'} : Bool;   // Head#3 manual jog forward fdbk {x|x|x|x|O}
            xManJogBackwardFdbk_H3 { ExternalWritable := 'False'} : Bool;   // Head#3 manual jog backward fdbk {x|x|x|x|O}
            xManJogForwardFdbk_H4 { ExternalWritable := 'False'} : Bool;   // Head#4 manual jog forward fdbk {x|x|x|x|O}
            xManJogBackwardFdbk_H4 { ExternalWritable := 'False'} : Bool;   // Head#4 manual jog backward fdbk {x|x|x|x|O}
            xManJogForwardFdbk_H5 { ExternalWritable := 'False'} : Bool;   // Head#5 manual jog forward fdbk {x|x|x|x|O}
            xManJogBackwardFdbk_H5 { ExternalWritable := 'False'} : Bool;   // Head#5 manual jog backward fdbk {x|x|x|x|O}
            xManJogForwardFdbk_H6 { ExternalWritable := 'False'} : Bool;   // Head#6 manual jog forward fdbk {x|x|x|x|O}
            xManJogBackwardFdbk_H6 { ExternalWritable := 'False'} : Bool;   // Head#6 manual jog backward fdbk {x|x|x|x|O}
            xManJogForwardFdbk_H7 { ExternalWritable := 'False'} : Bool;   // Head#7 manual jog forward fdbk {x|x|x|x|O}
            xManJogBackwardFdbk_H7 { ExternalWritable := 'False'} : Bool;   // Head#7 manual jog backward fdbk {x|x|x|x|O}
            xManJogForwardFdbk_H8 { ExternalWritable := 'False'} : Bool;   // Head#8 manual jog forward fdbk {x|x|x|x|O}
            xManJogBackwardFdbk_H8 { ExternalWritable := 'False'} : Bool;   // Head#8 manual jog backward fdbk {x|x|x|x|O}
            xSpare { ExternalWritable := 'False'} : Array[0..15] of Bool;
         END_STRUCT;
      END_STRUCT;
      tHMW : Struct   // HMI Write
         xBrakeRealeaseHead_H1 : Bool;   // Force the brake release of the Head #1 {x|x|x|x|M}
         xBrakeEngageHeads_H1 : Bool;   // Force the brake engaged of the Head #1 {x|x|x|x|M}
         xUpdateHomeHead_H1 : Bool;   // Update home position Head #1 {x|x|x|x|M}
         xBrakeRealeaseHead_H2 : Bool;   // Force the brake release of the Head #2 {x|x|x|x|M}
         xBrakeEngageHeads_H2 : Bool;   // Force the brake engaged of the Head #2 {x|x|x|x|M}
         xUpdateHomeHead_H2 : Bool;   // Update home position Head #2 {x|x|x|x|M}
         xBrakeRealeaseHead_H3 : Bool;   // Force the brake release of the Head #3 {x|x|x|x|M}
         xBrakeEngageHeads_H3 : Bool;   // Force the brake engaged of the Head #3 {x|x|x|x|M}
         xUpdateHomeHead_H3 : Bool;   // Update home position Head #3 {x|x|x|x|M}
         xBrakeRealeaseHead_H4 : Bool;   // Force the brake release of the Head #4{x|x|x|x|M}
         xBrakeEngageHeads_H4 : Bool;   // Force the brake engaged of the Head #4{x|x|x|x|M}
         xUpdateHomeHead_H4 : Bool;   // Update home position Head #4 {x|x|x|x|M}
         xBrakeRealeaseHead_H5 : Bool;   // Force the brake release of the Head #5{x|x|x|x|M}
         xBrakeEngageHeads_H5 : Bool;   // Force the brake engaged of the Head #5{x|x|x|x|M}
         xUpdateHomeHead_H5 : Bool;   // Update home position Head #5 {x|x|x|x|M}
         xBrakeRealeaseHead_H6 : Bool;   // Force the brake release of the Head #6{x|x|x|x|M}
         xBrakeEngageHeads_H6 : Bool;   // Force the brake engaged of the Head #6 {x|x|x|x|M}
         xUpdateHomeHead_H6 : Bool;   // Update home position Head #6 {x|x|x|x|M}
         xBrakeRealeaseHead_H7 : Bool;   // Force the brake release of the Head #7{x|x|x|x|M}
         xBrakeEngageHeads_H7 : Bool;   // Force the brake engaged of the Head #7{x|x|x|x|M}
         xUpdateHomeHead_H7 : Bool;   // Update home position Head #7{x|x|x|x|M}
         xBrakeRealeaseHead_H8 : Bool;   // Force the brake release of the Head #8{x|x|x|x|M}
         xBrakeEngageHeads_H8 : Bool;   // Force the brake engaged of the Head #8{x|x|x|x|M}
         xUpdateHomeHead_H8 : Bool;   // Update home position Head #8 {x|x|x|x|M}
         xSpare24 : Bool;
         xSpare25 : Bool;
         xSpare26 : Bool;
         xSpare27 : Bool;
         xSpare28 : Bool;
         xSpare29 : Bool;
         xSpare30 : Bool;
         xSpare31 : Bool;
         xSpare : Array[0..15] of Bool;
         iSpare0 : Int;
         iSpare1 : Int;
         iSpare2 : Int;
         iSpare3 : Int;
         iSpare4 : Int;
         iSpare5 : Int;
         iSpare6 : Int;
         iSpare7 : Int;
         iSpare8 : Int;
         iSpare9 : Int;
         iSpare10 : Int;
         iSpare11 : Int;
         iSpare12 : Int;
         iSpare13 : Int;
         iSpare14 : Int;
         iSpare15 : Int;
         iSpare16 : Int;
         dHeadHomePositions_cmm_H1 : DInt;   //  Head#1 home position [mm/100] {mm/100|mm|-2500|2500|M}
         dHeadHomePositions_cmm_H2 : DInt;   //  Head#2 home position [mm/100] {mm/100|mm|-2500|2500|M}
         dHeadHomePositions_cmm_H3 : DInt;   //  Head#3 home position [mm/100] {mm/100|mm|-2500|2500|M}
         dHeadHomePositions_cmm_H4 : DInt;   //  Head#4 home position [mm/100] {mm/100|mm|-2500|2500|M}
         dHeadHomePositions_cmm_H5 : DInt;   //  Head#5 home position [mm/100] {mm/100|mm|-2500|2500|M}
         dHeadHomePositions_cmm_H6 : DInt;   //  Head#6 home position [mm/100] {mm/100|mm|-2500|2500|M}
         dHeadHomePositions_cmm_H7 : DInt;   //  Head#7 home position [mm/100] {mm/100|mm|-2500|2500|M}
         dHeadHomePositions_cmm_H8 : DInt;   //  Head#8 home position [mm/100] {mm/100|mm|-2500|2500|M}
         dSpare8 : DInt;
         dSpare9 : DInt;
         dSpare10 : DInt;
         dSpare11 : DInt;
         dSpare12 : DInt;
         dSpare13 : DInt;
         dSpare14 : DInt;
         dSpare15 : DInt;
         dSpare { ExternalWritable := 'False'} : Array[0..43] of DInt;
         rSpare0 : Real;
         rSpare1 : Real;
         rSpare2 : Real;
         rSpare3 : Real;
         rSpare4 : Real;
         rSpare5 : Real;
         rSpare6 : Real;
         rSpare7 : Real;
         rSpare8 : Real;
         tManCmd : Struct
            xMan_JogForward_H1 : Bool;   // Head #1 manual jog forward {x|x|x|x|O}
            xMan_JogBackward_H1 : Bool;   // Head #1 manual jog backward {x|x|x|x|O}
            xMan_JogForward_H2 : Bool;   // Head #2 manual jog forward {x|x|x|x|O}
            xMan_JogBackward_H2 : Bool;   // Head #2 manual jog backward {x|x|x|x|O}
            xMan_JogForward_H3 : Bool;   // Head #3 manual jog forward {x|x|x|x|O}
            xMan_JogBackward_H3 : Bool;   // Head #3 manual jog backward {x|x|x|x|O}
            xMan_JogForward_H4 : Bool;   // Head #4 manual jog forward {x|x|x|x|O}
            xMan_JogBackward_H4 : Bool;   // Head #4 manual jog backward {x|x|x|x|O}
            xMan_JogForward_H5 : Bool;   // Head #5 manual jog forward {x|x|x|x|O}
            xMan_JogBackward_H5 : Bool;   // Head #5 manual jog backward {x|x|x|x|O}
            xMan_JogForward_H6 : Bool;   // Head #6 manual jog forward {x|x|x|x|O}
            xMan_JogBackward_H6 : Bool;   // Head #6 manual jog backward {x|x|x|x|O}
            xMan_JogForward_H7 : Bool;   // Head #7 manual jog forward {x|x|x|x|O}
            xMan_JogBackward_H7 : Bool;   // Head #7 manual jog backward {x|x|x|x|O}
            xMan_JogForward_H8 : Bool;   // Head #8 manual jog forward {x|x|x|x|O}
            xMan_JogBackward_H8 : Bool;   // Head #8 manual jog backward {x|x|x|x|O}
            xSpare16 : Bool;
            xSpare17 : Bool;
            xSpare18 : Bool;
            xSpare19 : Bool;
            xSpare20 : Bool;
            xSpare21 : Bool;
            xSpare22 : Bool;
            xSpare23 : Bool;
            xSpare24 : Bool;
            xSpare25 : Bool;
            xSpare26 : Bool;
            xSpare27 : Bool;
            xSpare28 : Bool;
            xSpare29 : Bool;
            xSpare30 : Bool;
            xSpare31 : Bool;
         END_STRUCT;
      END_STRUCT;
   END_STRUCT;


BEGIN
   tHMR.xSpare0 := FALSE;
   tHMR.xSpare15 := FALSE;
   tHMW.xBrakeRealeaseHead_H1 := FALSE;
   tHMW.xBrakeEngageHeads_H1 := FALSE;
   tHMW.xBrakeRealeaseHead_H2 := FALSE;
   tHMW.xBrakeEngageHeads_H2 := FALSE;
   tHMW.xBrakeRealeaseHead_H3 := FALSE;
   tHMW.xBrakeEngageHeads_H3 := FALSE;
   tHMW.xBrakeRealeaseHead_H4 := FALSE;
   tHMW.xBrakeEngageHeads_H4 := FALSE;
   tHMW.xBrakeRealeaseHead_H5 := FALSE;
   tHMW.xBrakeEngageHeads_H5 := FALSE;
   tHMW.xBrakeRealeaseHead_H6 := FALSE;
   tHMW.xBrakeEngageHeads_H6 := FALSE;
   tHMW.xBrakeRealeaseHead_H7 := FALSE;
   tHMW.xBrakeEngageHeads_H7 := FALSE;
   tHMW.xBrakeRealeaseHead_H8 := FALSE;
   tHMW.xBrakeEngageHeads_H8 := FALSE;

END_DATA_BLOCK

